LIN {X 0,Y 376.669,Z 402.869,A -85,B 0,C 180,E1 17335.147,E2 17335.147} C_VEL
LIN {X 0,Y 377.645,Z 382.714,A -85,B 0,C 180,E1 17334.66,E2 17334.66} C_VEL
LIN {X 0,Y 382.7,Z 216.459,A -85,B 0,C 180,E1 17331.601,E2 17331.601} C_VEL
LIN {X 0,Y 379.603,Z 196.687,A -85,B 0,C 180,E1 17330.72,E2 17330.72} C_VEL
LIN {X 0,Y 369.544,Z 178.657,A -85,B 0,C 180,E1 17328.838,E2 17328.838} C_VEL
LIN {X 0,Y 365.647,Z 171.977,A -85,B 0,C 180,E1 17328.055,E2 17328.055} C_VEL
LIN {X 0,Y 359.948,Z 157.351,A -85,B 0,C 180,E1 17324.899,E2 17324.899} C_VEL
LIN {X 0,Y 355.879,Z 147.74,A -85,B 0,C 180,E1 17322.598,E2 17322.598} C_VEL
LIN {X 0,Y 354.37,Z 147.289,A -85,B 0,C 180,E1 17322.197,E2 17322.197} C_VEL
LIN {X 0,Y 362.274,Z 168.365,A -85,B 0,C 180,E1 17319.144,E2 17319.144} C_VEL
LIN {X 0,Y 367.234,Z 183.559,A -85,B 0,C 180,E1 17317.084,E2 17317.084} C_VEL
LIN {X 0,Y 367.044,Z 189.046,A -85,B 0,C 180,E1 17316.607,E2 17316.607} C_VEL
LIN {X 0,Y 369.716,Z 213.655,A -85,B 0,C 180,E1 17315.636,E2 17315.636} C_VEL
LIN {X 0,Y 361.105,Z 400.958,A -85,B 0,C 180,E1 17310.874,E2 17310.874} C_VEL
LIN {X 0,Y 359.929,Z 421.052,A -85,B 0,C 180,E1 17310.048,E2 17310.048} C_VEL
LIN {X 0,Y 358.426,Z 440.427,A -85,B 0,C 180,E1 17308.947,E2 17308.947} C_VEL
LIN {X 0,Y 356.648,Z 459.281,A -85,B 0,C 180,E1 17307.554,E2 17307.554} C_VEL
LIN {X 0,Y 354.737,Z 477.04,A -85,B 0,C 180,E1 17305.905,E2 17305.905} C_VEL
LIN {X 0,Y 352.847,Z 493.012,A -85,B 0,C 180,E1 17304.083,E2 17304.083} C_VEL
LIN {X 0,Y 350.962,Z 507.993,A -85,B 0,C 180,E1 17302.002,E2 17302.002} C_VEL
LIN {X 0,Y 349.248,Z 521.455,A -85,B 0,C 180,E1 17299.745,E2 17299.745} C_VEL
LIN {X 0,Y 347.772,Z 533.32,A -85,B 0,C 180,E1 17297.345,E2 17297.345} C_VEL
LIN {X 0,Y 346.531,Z 544.028,A -85,B 0,C 180,E1 17294.709,E2 17294.709} C_VEL
LIN {X 0,Y 345.628,Z 552.855,A -85,B 0,C 180,E1 17292.022,E2 17292.022} C_VEL
LIN {X 0,Y 345.01,Z 560.233,A -85,B 0,C 180,E1 17289.172,E2 17289.172} C_VEL
LIN {X 0,Y 344.666,Z 565.763,A -85,B 0,C 180,E1 17286.329,E2 17286.329} C_VEL
LIN {X 0,Y 344.526,Z 569.587,A -85,B 0,C 180,E1 17283.494,E2 17283.494} C_VEL
LIN {X 0,Y 344.534,Z 571.796,A -85,B 0,C 180,E1 17280.665,E2 17280.665} C_VEL
LIN {X 0,Y 344.642,Z 572.453,A -85,B 0,C 180,E1 17277.839,E2 17277.839} C_VEL
LIN {X 0,Y 344.913,Z 571.551,A -85,B 0,C 180,E1 17275.011,E2 17275.011} C_VEL
LIN {X 0,Y 345.449,Z 568.896,A -85,B 0,C 180,E1 17272.014,E2 17272.014} C_VEL
LIN {X 0,Y 346.264,Z 564.713,A -85,B 0,C 180,E1 17269.182,E2 17269.182} C_VEL
LIN {X 0,Y 347.473,Z 558.782,A -85,B 0,C 180,E1 17266.352,E2 17266.352} C_VEL
LIN {X 0,Y 349.147,Z 550.97,A -85,B 0,C 180,E1 17263.531,E2 17263.531} C_VEL
LIN {X 0,Y 351.311,Z 540.92,A -85,B 0,C 180,E1 17260.723,E2 17260.723} C_VEL
LIN {X 0,Y 353.667,Z 529.913,A -85,B 0,C 180,E1 17258.263,E2 17258.263} C_VEL
LIN {X 0,Y 356.37,Z 517.049,A -85,B 0,C 180,E1 17255.907,E2 17255.907} C_VEL
LIN {X 0,Y 359.387,Z 501.97,A -85,B 0,C 180,E1 17253.657,E2 17253.657} C_VEL
LIN {X 0,Y 362.402,Z 485.474,A -85,B 0,C 180,E1 17251.671,E2 17251.671} C_VEL
LIN {X 0,Y 365.204,Z 468.627,A -85,B 0,C 180,E1 17250.023,E2 17250.023} C_VEL
LIN {X 0,Y 367.98,Z 450.12,A -85,B 0,C 180,E1 17248.554,E2 17248.554} C_VEL
LIN {X 0,Y 370.431,Z 430.981,A -85,B 0,C 180,E1 17247.368,E2 17247.368} C_VEL
LIN {X 0,Y 372.734,Z 409.425,A -85,B 0,C 180,E1 17246.363,E2 17246.363} C_VEL
LIN {X 0,Y 379.272,Z 352.203,A -85,B 0,C 180,E1 17244.383,E2 17244.383} C_VEL
LIN {X 0,Y 390.085,Z 279.328,A -85,B 0,C 180,E1 17241.833,E2 17241.833} C_VEL
LIN {X 0,Y 400.023,Z 222.705,A -85,B 0,C 180,E1 17239.855,E2 17239.855} C_VEL
LIN {X 0,Y 401.337,Z 211.185,A -85,B 0,C 180,E1 17238.798,E2 17238.798} C_VEL
LIN {X 0,Y 402.354,Z 207.214,A -85,B 0,C 180,E1 17238.338,E2 17238.338} C_VEL
LIN {X 0,Y 402.852,Z 202.964,A -85,B 0,C 180,E1 17236.862,E2 17236.862} C_VEL
LIN {X 0,Y 402.955,Z 202.336,A -85,B 0,C 180,E1 17236.432,E2 17236.432} C_VEL
LIN {X 0,Y 401.64,Z 206.111,A -85,B 0,C 180,E1 17235.499,E2 17235.499} C_VEL
LIN {X 0,Y 397.147,Z 221.02,A -85,B 0,C 180,E1 17234.85,E2 17234.85} C_VEL
LIN {X 0,Y 391.835,Z 244.614,A -85,B 0,C 180,E1 17234.018,E2 17234.018} C_VEL
LIN {X 0,Y 386.903,Z 267.436,A -85,B 0,C 180,E1 17233.236,E2 17233.236} C_VEL
LIN {X 0,Y 381.44,Z 294.492,A -85,B 0,C 180,E1 17232.25,E2 17232.25} C_VEL
LIN {X 0,Y 380.922,Z 302.139,A -85,B 0,C 180,E1 17232.058,E2 17232.058} C_VEL
LIN {X 0,Y 376.096,Z 417.535,A -85,B 0,C 180,E1 17229.641,E2 17229.641} C_VEL
LIN {X 0,Y 374.183,Z 439.175,A -85,B 0,C 180,E1 17228.934,E2 17228.934} C_VEL
LIN {X 0,Y 371.625,Z 460.279,A -85,B 0,C 180,E1 17227.947,E2 17227.947} C_VEL
LIN {X 0,Y 368.729,Z 479.932,A -85,B 0,C 180,E1 17226.722,E2 17226.722} C_VEL
LIN {X 0,Y 365.546,Z 498.613,A -85,B 0,C 180,E1 17225.25,E2 17225.25} C_VEL
LIN {X 0,Y 362.19,Z 516.529,A -85,B 0,C 180,E1 17223.513,E2 17223.513} C_VEL
LIN {X 0,Y 358.741,Z 533.822,A -85,B 0,C 180,E1 17221.476,E2 17221.476} C_VEL
LIN {X 0,Y 355.347,Z 550.311,A -85,B 0,C 180,E1 17219.13,E2 17219.13} C_VEL
LIN {X 0,Y 352.162,Z 565.804,A -85,B 0,C 180,E1 17216.473,E2 17216.473} C_VEL
LIN {X 0,Y 349.453,Z 579.625,A -85,B 0,C 180,E1 17213.615,E2 17213.615} C_VEL
LIN {X 0,Y 347.3,Z 591.834,A -85,B 0,C 180,E1 17210.564,E2 17210.564} C_VEL
LIN {X 0,Y 345.79,Z 601.923,A -85,B 0,C 180,E1 17207.502,E2 17207.502} C_VEL
LIN {X 0,Y 344.838,Z 610.17,A -85,B 0,C 180,E1 17204.436,E2 17204.436} C_VEL
LIN {X 0,Y 344.332,Z 616.936,A -85,B 0,C 180,E1 17201.22,E2 17201.22} C_VEL
LIN {X 0,Y 344.184,Z 621.714,A -85,B 0,C 180,E1 17198.185,E2 17198.185} C_VEL
LIN {X 0,Y 344.208,Z 625.148,A -85,B 0,C 180,E1 17195,E2 17195} C_VEL
LIN {X 0,Y 344.272,Z 626.894,A -85,B 0,C 180,E1 17191.998,E2 17191.998} C_VEL
LIN {X 0,Y 344.295,Z 627.095,A -85,B 0,C 180,E1 17189.003,E2 17189.003} C_VEL
LIN {X 0,Y 344.226,Z 625.768,A -85,B 0,C 180,E1 17185.837,E2 17185.837} C_VEL
LIN {X 0,Y 344.176,Z 623.016,A -85,B 0,C 180,E1 17182.825,E2 17182.825} C_VEL
LIN {X 0,Y 344.265,Z 618.402,A -85,B 0,C 180,E1 17179.627,E2 17179.627} C_VEL
LIN {X 0,Y 344.668,Z 611.955,A -85,B 0,C 180,E1 17176.363,E2 17176.363} C_VEL
LIN {X 0,Y 345.594,Z 603.383,A -85,B 0,C 180,E1 17173.011,E2 17173.011} C_VEL
LIN {X 0,Y 347.008,Z 593.607,A -85,B 0,C 180,E1 17169.938,E2 17169.938} C_VEL
LIN {X 0,Y 348.916,Z 582.559,A -85,B 0,C 180,E1 17167.064,E2 17167.064} C_VEL
LIN {X 0,Y 351.468,Z 569.316,A -85,B 0,C 180,E1 17164.2,E2 17164.2} C_VEL
LIN {X 0,Y 354.48,Z 554.472,A -85,B 0,C 180,E1 17161.532,E2 17161.532} C_VEL
LIN {X 0,Y 357.942,Z 537.753,A -85,B 0,C 180,E1 17159.043,E2 17159.043} C_VEL
LIN {X 0,Y 361.466,Z 520.196,A -85,B 0,C 180,E1 17156.887,E2 17156.887} C_VEL
LIN {X 0,Y 364.9,Z 502.06,A -85,B 0,C 180,E1 17155.064,E2 17155.064} C_VEL
LIN {X 0,Y 368.013,Z 483.999,A -85,B 0,C 180,E1 17153.585,E2 17153.585} C_VEL
LIN {X 0,Y 370.849,Z 465.441,A -85,B 0,C 180,E1 17152.363,E2 17152.363} C_VEL
LIN {X 0,Y 373.499,Z 444.639,A -85,B 0,C 180,E1 17151.307,E2 17151.307} C_VEL
LIN {X 0,Y 375.593,Z 423.414,A -85,B 0,C 180,E1 17150.54,E2 17150.54} C_VEL
LIN {X 0,Y 376.937,Z 399.024,A -85,B 0,C 180,E1 17149.951,E2 17149.951} C_VEL
LIN {X 0,Y 384.948,Z 202.452,A -85,B 0,C 180,E1 17145.917,E2 17145.917} C_VEL
LIN {X 0,Y 384.473,Z 199.885,A -85,B 0,C 180,E1 17145.79,E2 17145.79} C_VEL
LIN {X 0,Y 373.483,Z 180.271,A -85,B 0,C 180,E1 17143.765,E2 17143.765} C_VEL
LIN {X 0,Y 364.515,Z 165.595,A -85,B 0,C 180,E1 17141.984,E2 17141.984} C_VEL
LIN {X 0,Y 358.147,Z 151.33,A -85,B 0,C 180,E1 17138.913,E2 17138.913} C_VEL
LIN {X 0,Y 352.636,Z 139.889,A -85,B 0,C 180,E1 17136.14,E2 17136.14} C_VEL
LIN {X 0,Y 350.054,Z 135.087,A -85,B 0,C 180,E1 17134.838,E2 17134.838} C_VEL
LIN {X 0,Y 347.982,Z 130.852,A -85,B 0,C 180,E1 17133.679,E2 17133.679} C_VEL
LIN {X 0,Y 346.134,Z 127.573,A -85,B 0,C 180,E1 17132.695,E2 17132.695} C_VEL
LIN {X 0,Y 345.909,Z 126.377,A -85,B 0,C 180,E1 17132.38,E2 17132.38} C_VEL
LIN {X 0,Y 345.922,Z 126.373,A -85,B 0,C 180,E1 17128.17,E2 17128.17} C_VEL
LIN {X 0,Y 345.893,Z 126.372,A -85,B 0,C 180,E1 17123.871,E2 17123.871} C_VEL
LIN {X 0,Y 345.886,Z 126.376,A -85,B 0,C 180,E1 17119.768,E2 17119.768} C_VEL
LIN {X 0,Y 345.877,Z 126.4,A -85,B 0,C 180,E1 17115.595,E2 17115.595} C_VEL
LIN {X 0,Y 345.872,Z 126.388,A -85,B 0,C 180,E1 17111.337,E2 17111.337} C_VEL
LIN {X 0,Y 345.87,Z 126.366,A -85,B 0,C 180,E1 17107.14,E2 17107.14} C_VEL
LIN {X 0,Y 345.88,Z 126.39,A -85,B 0,C 180,E1 17102.982,E2 17102.982} C_VEL
LIN {X 0,Y 345.886,Z 126.391,A -85,B 0,C 180,E1 17098.84,E2 17098.84} C_VEL
LIN {X 0,Y 345.892,Z 126.363,A -85,B 0,C 180,E1 17094.692,E2 17094.692} C_VEL
LIN {X 0,Y 345.902,Z 126.39,A -85,B 0,C 180,E1 17090.516,E2 17090.516} C_VEL
LIN {X 0,Y 345.89,Z 126.392,A -85,B 0,C 180,E1 17086.227,E2 17086.227} C_VEL
LIN {X 0,Y 345.881,Z 126.368,A -85,B 0,C 180,E1 17082.156,E2 17082.156} C_VEL
LIN {X 0,Y 345.868,Z 126.38,A -85,B 0,C 180,E1 17077.925,E2 17077.925} C_VEL
LIN {X 0,Y 345.865,Z 126.4,A -85,B 0,C 180,E1 17073.657,E2 17073.657} C_VEL
LIN {X 0,Y 345.863,Z 126.401,A -85,B 0,C 180,E1 17069.416,E2 17069.416} C_VEL
LIN {X 0,Y 345.875,Z 126.395,A -85,B 0,C 180,E1 17065.182,E2 17065.182} C_VEL
LIN {X 0,Y 345.905,Z 126.617,A -85,B 0,C 180,E1 17063.193,E2 17063.193} C_VEL
LIN {X 0,Y 347.343,Z 130.105,A -85,B 0,C 180,E1 17062.183,E2 17062.183} C_VEL
LIN {X 0,Y 348.365,Z 132.049,A -85,B 0,C 180,E1 17061.585,E2 17061.585} C_VEL
LIN {X 0,Y 350.531,Z 136.549,A -85,B 0,C 180,E1 17060.287,E2 17060.287} C_VEL
LIN {X 0,Y 354.726,Z 145.516,A -85,B 0,C 180,E1 17057.867,E2 17057.867} C_VEL
LIN {X 0,Y 360.366,Z 158.402,A -85,B 0,C 180,E1 17054.741,E2 17054.741} C_VEL
LIN {X 0,Y 365.903,Z 172.565,A -85,B 0,C 180,E1 17051.755,E2 17051.755} C_VEL
LIN {X 0,Y 376.444,Z 190.872,A -85,B 0,C 180,E1 17049.742,E2 17049.742} C_VEL
LIN {X 0,Y 379.861,Z 197.758,A -85,B 0,C 180,E1 17049.104,E2 17049.104} C_VEL
LIN {X 0,Y 382.711,Z 218.275,A -85,B 0,C 180,E1 17048.246,E2 17048.246} C_VEL
LIN {X 0,Y 377.126,Z 394.489,A -85,B 0,C 180,E1 17044.986,E2 17044.986} C_VEL
LIN {X 0,Y 375.738,Z 413.928,A -85,B 0,C 180,E1 17044.359,E2 17044.359} C_VEL
LIN {X 0,Y 373.878,Z 431.784,A -85,B 0,C 180,E1 17043.52,E2 17043.52} C_VEL
LIN {X 0,Y 371.403,Z 449.716,A -85,B 0,C 180,E1 17042.392,E2 17042.392} C_VEL
LIN {X 0,Y 368.525,Z 466.63,A -85,B 0,C 180,E1 17041.029,E2 17041.029} C_VEL
LIN {X 0,Y 365.237,Z 483.324,A -85,B 0,C 180,E1 17039.341,E2 17039.341} C_VEL
LIN {X 0,Y 361.781,Z 498.814,A -85,B 0,C 180,E1 17037.396,E2 17037.396} C_VEL
LIN {X 0,Y 358.417,Z 512.658,A -85,B 0,C 180,E1 17035.264,E2 17035.264} C_VEL
LIN {X 0,Y 355.163,Z 525.427,A -85,B 0,C 180,E1 17032.86,E2 17032.86} C_VEL
LIN {X 0,Y 352.22,Z 536.673,A -85,B 0,C 180,E1 17030.261,E2 17030.261} C_VEL
LIN {X 0,Y 349.57,Z 546.939,A -85,B 0,C 180,E1 17027.304,E2 17027.304} C_VEL
LIN {X 0,Y 347.575,Z 555.103,A -85,B 0,C 180,E1 17024.322,E2 17024.322} C_VEL
LIN {X 0,Y 346.111,Z 561.733,A -85,B 0,C 180,E1 17021.159,E2 17021.159} C_VEL
LIN {X 0,Y 345.205,Z 566.551,A -85,B 0,C 180,E1 17017.99,E2 17017.99} C_VEL
LIN {X 0,Y 344.718,Z 569.704,A -85,B 0,C 180,E1 17014.824,E2 17014.824} C_VEL
LIN {X 0,Y 344.514,Z 571.318,A -85,B 0,C 180,E1 17011.496,E2 17011.496} C_VEL
LIN {X 0,Y 344.523,Z 571.26,A -85,B 0,C 180,E1 17008.17,E2 17008.17} C_VEL
LIN {X 0,Y 344.742,Z 569.524,A -85,B 0,C 180,E1 17004.841,E2 17004.841} C_VEL
LIN {X 0,Y 345.047,Z 567.492,A -85,B 0,C 180,E1 17002.726,E2 17002.726} C_VEL
LIN {X 0,Y 344.31,Z 566.093,A -85,B 0,C 180,E1 17001.465,E2 17001.465} C_VEL
LIN {X 0,Y 339.153,Z 561.593,A -85,B 0,C 180,E1 16998.087,E2 16998.087} C_VEL
LIN {X 0,Y 338.885,Z 559.609,A -85,B 0,C 180,E1 16997.007,E2 16997.007} C_VEL
LIN {X 0,Y 340.728,Z 552.186,A -85,B 0,C 180,E1 16993.812,E2 16993.812} C_VEL
LIN {X 0,Y 343.148,Z 543.092,A -85,B 0,C 180,E1 16990.775,E2 16990.775} C_VEL
LIN {X 0,Y 346.088,Z 532.413,A -85,B 0,C 180,E1 16987.939,E2 16987.939} C_VEL
LIN {X 0,Y 349.449,Z 520.13,A -85,B 0,C 180,E1 16985.307,E2 16985.307} C_VEL
LIN {X 0,Y 352.96,Z 506.734,A -85,B 0,C 180,E1 16982.974,E2 16982.974} C_VEL
LIN {X 0,Y 356.567,Z 492.027,A -85,B 0,C 180,E1 16980.887,E2 16980.887} C_VEL
LIN {X 0,Y 360.18,Z 475.636,A -85,B 0,C 180,E1 16979.005,E2 16979.005} C_VEL
LIN {X 0,Y 363.415,Z 458.807,A -85,B 0,C 180,E1 16977.46,E2 16977.46} C_VEL
LIN {X 0,Y 366.3,Z 440.809,A -85,B 0,C 180,E1 16976.161,E2 16976.161} C_VEL
LIN {X 0,Y 368.645,Z 422.047,A -85,B 0,C 180,E1 16975.137,E2 16975.137} C_VEL
LIN {X 0,Y 370.332,Z 403.037,A -85,B 0,C 180,E1 16974.396,E2 16974.396} C_VEL
LIN {X 0,Y 371.349,Z 382.958,A -85,B 0,C 180,E1 16973.905,E2 16973.905} C_VEL
LIN {X 0,Y 376.667,Z 217.846,A -85,B 0,C 180,E1 16970.825,E2 16970.825} C_VEL
LIN {X 0,Y 374.047,Z 200.618,A -85,B 0,C 180,E1 16970.042,E2 16970.042} C_VEL
LIN {X 0,Y 363.82,Z 182.148,A -85,B 0,C 180,E1 16968.051,E2 16968.051} C_VEL
LIN {X 0,Y 357.676,Z 171.867,A -85,B 0,C 180,E1 16966.773,E2 16966.773} C_VEL
LIN {X 0,Y 351.569,Z 156.622,A -85,B 0,C 180,E1 16963.268,E2 16963.268} C_VEL
LIN {X 0,Y 350.226,Z 154.037,A -85,B 0,C 180,E1 16962.58,E2 16962.58} C_VEL
LIN {X 0,Y 348.669,Z 153.653,A -85,B 0,C 180,E1 16962.158,E2 16962.158} C_VEL
LIN {X 0,Y 356.203,Z 174.193,A -85,B 0,C 180,E1 16959.167,E2 16959.167} C_VEL
LIN {X 0,Y 360.109,Z 185.882,A -85,B 0,C 180,E1 16957.56,E2 16957.56} C_VEL
LIN {X 0,Y 360.055,Z 189.639,A -85,B 0,C 180,E1 16957.242,E2 16957.242} C_VEL
LIN {X 0,Y 362.693,Z 214.583,A -85,B 0,C 180,E1 16956.227,E2 16956.227} C_VEL
LIN {X 0,Y 353.679,Z 401.543,A -85,B 0,C 180,E1 16951.344,E2 16951.344} C_VEL
LIN {X 0,Y 352.479,Z 421.326,A -85,B 0,C 180,E1 16950.515,E2 16950.515} C_VEL
LIN {X 0,Y 350.98,Z 440.119,A -85,B 0,C 180,E1 16949.434,E2 16949.434} C_VEL
LIN {X 0,Y 349.131,Z 459.141,A -85,B 0,C 180,E1 16948.013,E2 16948.013} C_VEL
LIN {X 0,Y 347.255,Z 476.075,A -85,B 0,C 180,E1 16946.43,E2 16946.43} C_VEL
LIN {X 0,Y 345.316,Z 492.049,A -85,B 0,C 180,E1 16944.605,E2 16944.605} C_VEL
LIN {X 0,Y 343.374,Z 507.168,A -85,B 0,C 180,E1 16942.514,E2 16942.514} C_VEL
LIN {X 0,Y 341.566,Z 520.911,A -85,B 0,C 180,E1 16940.208,E2 16940.208} C_VEL
LIN {X 0,Y 340.033,Z 532.774,A -85,B 0,C 180,E1 16937.807,E2 16937.807} C_VEL
LIN {X 0,Y 338.725,Z 543.603,A -85,B 0,C 180,E1 16935.146,E2 16935.146} C_VEL
LIN {X 0,Y 337.728,Z 552.932,A -85,B 0,C 180,E1 16932.308,E2 16932.308} C_VEL
LIN {X 0,Y 337.065,Z 560.461,A -85,B 0,C 180,E1 16929.39,E2 16929.39} C_VEL
LIN {X 0,Y 336.697,Z 566.123,A -85,B 0,C 180,E1 16926.48,E2 16926.48} C_VEL
LIN {X 0,Y 336.547,Z 570.075,A -85,B 0,C 180,E1 16923.577,E2 16923.577} C_VEL
LIN {X 0,Y 336.558,Z 572.419,A -85,B 0,C 180,E1 16920.681,E2 16920.681} C_VEL
LIN {X 0,Y 336.679,Z 573.197,A -85,B 0,C 180,E1 16917.788,E2 16917.788} C_VEL
LIN {X 0,Y 336.979,Z 572.412,A -85,B 0,C 180,E1 16914.893,E2 16914.893} C_VEL
LIN {X 0,Y 337.566,Z 569.88,A -85,B 0,C 180,E1 16911.827,E2 16911.827} C_VEL
LIN {X 0,Y 338.522,Z 565.528,A -85,B 0,C 180,E1 16908.759,E2 16908.759} C_VEL
LIN {X 0,Y 339.865,Z 559.637,A -85,B 0,C 180,E1 16905.867,E2 16905.867} C_VEL
LIN {X 0,Y 341.702,Z 551.853,A -85,B 0,C 180,E1 16902.986,E2 16902.986} C_VEL
LIN {X 0,Y 343.909,Z 542.508,A -85,B 0,C 180,E1 16900.291,E2 16900.291} C_VEL
LIN {X 0,Y 346.448,Z 531.764,A -85,B 0,C 180,E1 16897.786,E2 16897.786} C_VEL
LIN {X 0,Y 349.439,Z 518.656,A -85,B 0,C 180,E1 16895.307,E2 16895.307} C_VEL
LIN {X 0,Y 352.669,Z 503.818,A -85,B 0,C 180,E1 16893.024,E2 16893.024} C_VEL
LIN {X 0,Y 355.777,Z 488.46,A -85,B 0,C 180,E1 16891.094,E2 16891.094} C_VEL
LIN {X 0,Y 358.924,Z 471.463,A -85,B 0,C 180,E1 16889.351,E2 16889.351} C_VEL
LIN {X 0,Y 362.057,Z 452.668,A -85,B 0,C 180,E1 16887.793,E2 16887.793} C_VEL
LIN {X 0,Y 364.883,Z 433.34,A -85,B 0,C 180,E1 16886.532,E2 16886.532} C_VEL
LIN {X 0,Y 367.478,Z 411.855,A -85,B 0,C 180,E1 16885.479,E2 16885.479} C_VEL
LIN {X 0,Y 374.158,Z 359.163,A -85,B 0,C 180,E1 16883.577,E2 16883.577} C_VEL
LIN {X 0,Y 385.505,Z 288.757,A -85,B 0,C 180,E1 16881.051,E2 16881.051} C_VEL
LIN {X 0,Y 397.659,Z 225.322,A -85,B 0,C 180,E1 16878.807,E2 16878.807} C_VEL
LIN {X 0,Y 399.563,Z 213.082,A -85,B 0,C 180,E1 16877.631,E2 16877.631} C_VEL
LIN {X 0,Y 400.105,Z 210.398,A -85,B 0,C 180,E1 16876.607,E2 16876.607} C_VEL
LIN {X 0,Y 399.764,Z 211.263,A -85,B 0,C 180,E1 16876.445,E2 16876.445} C_VEL
LIN {X 0,Y 396.708,Z 221.504,A -85,B 0,C 180,E1 16876.033,E2 16876.033} C_VEL
LIN {X 0,Y 389.126,Z 252.716,A -85,B 0,C 180,E1 16874.961,E2 16874.961} C_VEL
LIN {X 0,Y 383.159,Z 278.56,A -85,B 0,C 180,E1 16874.05,E2 16874.05} C_VEL
LIN {X 0,Y 377.866,Z 302.725,A -85,B 0,C 180,E1 16873.172,E2 16873.172} C_VEL
LIN {X 0,Y 373.832,Z 323.539,A -85,B 0,C 180,E1 16872.388,E2 16872.388} C_VEL
LIN {X 0,Y 369.736,Z 417.309,A -85,B 0,C 180,E1 16870.392,E2 16870.392} C_VEL
LIN {X 0,Y 367.763,Z 438.86,A -85,B 0,C 180,E1 16869.68,E2 16869.68} C_VEL
LIN {X 0,Y 365.152,Z 459.562,A -85,B 0,C 180,E1 16868.704,E2 16868.704} C_VEL
LIN {X 0,Y 362.026,Z 479.974,A -85,B 0,C 180,E1 16867.418,E2 16867.418} C_VEL
LIN {X 0,Y 358.545,Z 499.478,A -85,B 0,C 180,E1 16865.848,E2 16865.848} C_VEL
LIN {X 0,Y 354.905,Z 517.907,A -85,B 0,C 180,E1 16864.003,E2 16864.003} C_VEL
LIN {X 0,Y 351.368,Z 534.672,A -85,B 0,C 180,E1 16861.958,E2 16861.958} C_VEL
LIN {X 0,Y 347.911,Z 550.579,A -85,B 0,C 180,E1 16859.625,E2 16859.625} C_VEL
LIN {X 0,Y 344.755,Z 565.071,A -85,B 0,C 180,E1 16857.082,E2 16857.082} C_VEL
LIN {X 0,Y 341.855,Z 579.016,A -85,B 0,C 180,E1 16854.142,E2 16854.142} C_VEL
LIN {X 0,Y 339.553,Z 591.234,A -85,B 0,C 180,E1 16851.022,E2 16851.022} C_VEL
LIN {X 0,Y 337.943,Z 601.228,A -85,B 0,C 180,E1 16847.922,E2 16847.922} C_VEL
LIN {X 0,Y 336.878,Z 609.823,A -85,B 0,C 180,E1 16844.632,E2 16844.632} C_VEL
LIN {X 0,Y 336.343,Z 616.593,A -85,B 0,C 180,E1 16841.316,E2 16841.316} C_VEL
LIN {X 0,Y 336.193,Z 621.506,A -85,B 0,C 180,E1 16838.036,E2 16838.036} C_VEL
LIN {X 0,Y 336.232,Z 624.749,A -85,B 0,C 180,E1 16834.777,E2 16834.777} C_VEL
LIN {X 0,Y 336.303,Z 626.347,A -85,B 0,C 180,E1 16831.705,E2 16831.705} C_VEL
LIN {X 0,Y 336.317,Z 626.424,A -85,B 0,C 180,E1 16828.809,E2 16828.809} C_VEL
LIN {X 0,Y 336.24,Z 624.994,A -85,B 0,C 180,E1 16825.567,E2 16825.567} C_VEL
LIN {X 0,Y 336.187,Z 622.17,A -85,B 0,C 180,E1 16822.482,E2 16822.482} C_VEL
LIN {X 0,Y 336.301,Z 617.458,A -85,B 0,C 180,E1 16819.206,E2 16819.206} C_VEL
LIN {X 0,Y 336.755,Z 611,A -85,B 0,C 180,E1 16815.91,E2 16815.91} C_VEL
LIN {X 0,Y 337.734,Z 602.686,A -85,B 0,C 180,E1 16812.603,E2 16812.603} C_VEL
LIN {X 0,Y 339.356,Z 592.318,A -85,B 0,C 180,E1 16809.296,E2 16809.296} C_VEL
LIN {X 0,Y 341.442,Z 581.082,A -85,B 0,C 180,E1 16806.349,E2 16806.349} C_VEL
LIN {X 0,Y 344.14,Z 567.986,A -85,B 0,C 180,E1 16803.49,E2 16803.49} C_VEL
LIN {X 0,Y 347.337,Z 553.164,A -85,B 0,C 180,E1 16800.797,E2 16800.797} C_VEL
LIN {X 0,Y 350.834,Z 537.114,A -85,B 0,C 180,E1 16798.374,E2 16798.374} C_VEL
LIN {X 0,Y 354.597,Z 519.321,A -85,B 0,C 180,E1 16796.16,E2 16796.16} C_VEL
LIN {X 0,Y 358.364,Z 500.272,A -85,B 0,C 180,E1 16794.233,E2 16794.233} C_VEL
LIN {X 0,Y 361.828,Z 480.911,A -85,B 0,C 180,E1 16792.661,E2 16792.661} C_VEL
LIN {X 0,Y 364.803,Z 461.647,A -85,B 0,C 180,E1 16791.427,E2 16791.427} C_VEL
LIN {X 0,Y 367.379,Z 441.543,A -85,B 0,C 180,E1 16790.444,E2 16790.444} C_VEL
LIN {X 0,Y 369.386,Z 421.025,A -85,B 0,C 180,E1 16789.727,E2 16789.727} C_VEL
LIN {X 0,Y 370.89,Z 392.105,A -85,B 0,C 180,E1 16789.055,E2 16789.055} C_VEL
LIN {X 0,Y 378.87,Z 203.932,A -85,B 0,C 180,E1 16785.146,E2 16785.146} C_VEL
LIN {X 0,Y 368.573,Z 185.369,A -85,B 0,C 180,E1 16783.18,E2 16783.18} C_VEL
LIN {X 0,Y 358.66,Z 169.273,A -85,B 0,C 180,E1 16781.167,E2 16781.167} C_VEL
LIN {X 0,Y 356.331,Z 165.47,A -85,B 0,C 180,E1 16780.616,E2 16780.616} C_VEL
LIN {X 0,Y 350.756,Z 153.122,A -85,B 0,C 180,E1 16777.797,E2 16777.797} C_VEL
LIN {X 0,Y 345.132,Z 141.448,A -85,B 0,C 180,E1 16774.8,E2 16774.8} C_VEL
LIN {X 0,Y 342.33,Z 136.309,A -85,B 0,C 180,E1 16773.305,E2 16773.305} C_VEL
LIN {X 0,Y 340.529,Z 132.462,A -85,B 0,C 180,E1 16772.203,E2 16772.203} C_VEL
LIN {X 0,Y 338.247,Z 128.784,A -85,B 0,C 180,E1 16770.953,E2 16770.953} C_VEL
LIN {X 0,Y 337.961,Z 127.386,A -85,B 0,C 180,E1 16770.582,E2 16770.582} C_VEL
LIN {X 0,Y 337.974,Z 127.388,A -85,B 0,C 180,E1 16766.315,E2 16766.315} C_VEL
LIN {X 0,Y 337.97,Z 127.379,A -85,B 0,C 180,E1 16762.068,E2 16762.068} C_VEL
LIN {X 0,Y 337.944,Z 127.364,A -85,B 0,C 180,E1 16757.742,E2 16757.742} C_VEL
LIN {X 0,Y 337.934,Z 127.356,A -85,B 0,C 180,E1 16753.517,E2 16753.517} C_VEL
LIN {X 0,Y 337.935,Z 127.38,A -85,B 0,C 180,E1 16749.193,E2 16749.193} C_VEL
LIN {X 0,Y 337.944,Z 127.383,A -85,B 0,C 180,E1 16744.922,E2 16744.922} C_VEL
LIN {X 0,Y 337.962,Z 127.35,A -85,B 0,C 180,E1 16740.593,E2 16740.593} C_VEL
LIN {X 0,Y 337.96,Z 127.372,A -85,B 0,C 180,E1 16736.438,E2 16736.438} C_VEL
LIN {X 0,Y 337.952,Z 127.383,A -85,B 0,C 180,E1 16732.178,E2 16732.178} C_VEL
LIN {X 0,Y 337.932,Z 127.357,A -85,B 0,C 180,E1 16727.873,E2 16727.873} C_VEL
LIN {X 0,Y 337.926,Z 127.368,A -85,B 0,C 180,E1 16723.675,E2 16723.675} C_VEL
LIN {X 0,Y 337.93,Z 127.391,A -85,B 0,C 180,E1 16719.384,E2 16719.384} C_VEL
LIN {X 0,Y 337.934,Z 127.373,A -85,B 0,C 180,E1 16715.156,E2 16715.156} C_VEL
LIN {X 0,Y 337.945,Z 127.36,A -85,B 0,C 180,E1 16710.973,E2 16710.973} C_VEL
LIN {X 0,Y 337.951,Z 127.362,A -85,B 0,C 180,E1 16706.815,E2 16706.815} C_VEL
LIN {X 0,Y 337.979,Z 127.626,A -85,B 0,C 180,E1 16704.976,E2 16704.976} C_VEL
LIN {X 0,Y 339.396,Z 131.102,A -85,B 0,C 180,E1 16703.899,E2 16703.899} C_VEL
LIN {X 0,Y 340.451,Z 132.811,A -85,B 0,C 180,E1 16703.297,E2 16703.297} C_VEL
LIN {X 0,Y 344.764,Z 141.822,A -85,B 0,C 180,E1 16700.57,E2 16700.57} C_VEL
LIN {X 0,Y 349.842,Z 152.762,A -85,B 0,C 180,E1 16697.585,E2 16697.585} C_VEL
LIN {X 0,Y 355.683,Z 166.992,A -85,B 0,C 180,E1 16694.197,E2 16694.197} C_VEL
LIN {X 0,Y 357.902,Z 172.461,A -85,B 0,C 180,E1 16693.038,E2 16693.038} C_VEL
LIN {X 0,Y 368.613,Z 190.696,A -85,B 0,C 180,E1 16690.877,E2 16690.877} C_VEL
LIN {X 0,Y 374.224,Z 201.393,A -85,B 0,C 180,E1 16689.797,E2 16689.797} C_VEL
LIN {X 0,Y 376.663,Z 219.69,A -85,B 0,C 180,E1 16689.02,E2 16689.02} C_VEL
LIN {X 0,Y 370.794,Z 394.883,A -85,B 0,C 180,E1 16685.733,E2 16685.733} C_VEL
LIN {X 0,Y 369.349,Z 414.285,A -85,B 0,C 180,E1 16685.098,E2 16685.098} C_VEL
LIN {X 0,Y 367.3,Z 432.961,A -85,B 0,C 180,E1 16684.202,E2 16684.202} C_VEL
LIN {X 0,Y 364.727,Z 450.731,A -85,B 0,C 180,E1 16683.06,E2 16683.06} C_VEL
LIN {X 0,Y 361.572,Z 468.366,A -85,B 0,C 180,E1 16681.601,E2 16681.601} C_VEL
LIN {X 0,Y 358.159,Z 484.804,A -85,B 0,C 180,E1 16679.887,E2 16679.887} C_VEL
LIN {X 0,Y 354.57,Z 500.118,A -85,B 0,C 180,E1 16677.91,E2 16677.91} C_VEL
LIN {X 0,Y 351.2,Z 513.393,A -85,B 0,C 180,E1 16675.821,E2 16675.821} C_VEL
LIN {X 0,Y 347.793,Z 526.134,A -85,B 0,C 180,E1 16673.373,E2 16673.373} C_VEL
LIN {X 0,Y 344.705,Z 537.363,A -85,B 0,C 180,E1 16670.723,E2 16670.723} C_VEL
LIN {X 0,Y 342.053,Z 547.116,A -85,B 0,C 180,E1 16667.873,E2 16667.873} C_VEL
LIN {X 0,Y 339.906,Z 555.38,A -85,B 0,C 180,E1 16664.827,E2 16664.827} C_VEL
LIN {X 0,Y 338.317,Z 562.106,A -85,B 0,C 180,E1 16661.592,E2 16661.592} C_VEL
LIN {X 0,Y 337.323,Z 567.008,A -85,B 0,C 180,E1 16658.35,E2 16658.35} C_VEL
LIN {X 0,Y 336.76,Z 570.351,A -85,B 0,C 180,E1 16654.938,E2 16654.938} C_VEL
LIN {X 0,Y 336.541,Z 571.964,A -85,B 0,C 180,E1 16651.531,E2 16651.531} C_VEL
LIN {X 0,Y 336.551,Z 571.905,A -85,B 0,C 180,E1 16648.126,E2 16648.126} C_VEL
LIN {X 0,Y 336.787,Z 570.171,A -85,B 0,C 180,E1 16644.718,E2 16644.718} C_VEL
LIN {X 0,Y 337.344,Z 566.922,A -85,B 0,C 180,E1 16641.477,E2 16641.477} C_VEL
LIN {X 0,Y 338.42,Z 561.658,A -85,B 0,C 180,E1 16638.063,E2 16638.063} C_VEL
LIN {X 0,Y 338.885,Z 559.609,A -85,B 0,C 180,E1 16637.007,E2 16637.007} C_VEL
LIN {X 0,Y 338.544,Z 557.217,A -85,B 0,C 180,E1 16635.758,E2 16635.758} C_VEL
LIN {X 0,Y 334.79,Z 550.945,A -85,B 0,C 180,E1 16632.765,E2 16632.765} C_VEL
LIN {X 0,Y 334.502,Z 547.665,A -85,B 0,C 180,E1 16631.558,E2 16631.558} C_VEL
LIN {X 0,Y 334.618,Z 547.147,A -85,B 0,C 180,E1 16631.391,E2 16631.391} C_VEL
LIN {X 0,Y 337.5,Z 537.117,A -85,B 0,C 180,E1 16628.446,E2 16628.446} C_VEL
LIN {X 0,Y 340.799,Z 525.71,A -85,B 0,C 180,E1 16625.748,E2 16625.748} C_VEL
LIN {X 0,Y 344.423,Z 512.758,A -85,B 0,C 180,E1 16623.258,E2 16623.258} C_VEL
LIN {X 0,Y 348.132,Z 498.713,A -85,B 0,C 180,E1 16621.056,E2 16621.056} C_VEL
LIN {X 0,Y 351.771,Z 483.716,A -85,B 0,C 180,E1 16619.137,E2 16619.137} C_VEL
LIN {X 0,Y 355.2,Z 467.72,A -85,B 0,C 180,E1 16617.475,E2 16617.475} C_VEL
LIN {X 0,Y 358.319,Z 450.85,A -85,B 0,C 180,E1 16616.076,E2 16616.076} C_VEL
LIN {X 0,Y 361.089,Z 432.312,A -85,B 0,C 180,E1 16614.881,E2 16614.881} C_VEL
LIN {X 0,Y 363.233,Z 413.203,A -85,B 0,C 180,E1 16613.975,E2 16613.975} C_VEL
LIN {X 0,Y 364.676,Z 393.727,A -85,B 0,C 180,E1 16613.351,E2 16613.351} C_VEL
LIN {X 0,Y 370.694,Z 219.152,A -85,B 0,C 180,E1 16610.02,E2 16610.02} C_VEL
LIN {X 0,Y 368.466,Z 204.357,A -85,B 0,C 180,E1 16609.328,E2 16609.328} C_VEL
LIN {X 0,Y 358.773,Z 186.808,A -85,B 0,C 180,E1 16607.37,E2 16607.37} C_VEL
LIN {X 0,Y 349.655,Z 171.823,A -85,B 0,C 180,E1 16605.401,E2 16605.401} C_VEL
LIN {X 0,Y 345.002,Z 160.411,A -85,B 0,C 180,E1 16602.644,E2 16602.644} C_VEL
LIN {X 0,Y 342.949,Z 160.049,A -85,B 0,C 180,E1 16602.129,E2 16602.129} C_VEL
LIN {X 0,Y 350.82,Z 182.032,A -85,B 0,C 180,E1 16598.915,E2 16598.915} C_VEL
LIN {X 0,Y 352.984,Z 189.385,A -85,B 0,C 180,E1 16597.929,E2 16597.929} C_VEL
LIN {X 0,Y 355.682,Z 215.64,A -85,B 0,C 180,E1 16596.832,E2 16596.832} C_VEL
LIN {X 0,Y 346.28,Z 402.045,A -85,B 0,C 180,E1 16591.837,E2 16591.837} C_VEL
LIN {X 0,Y 345.051,Z 421.535,A -85,B 0,C 180,E1 16591.002,E2 16591.002} C_VEL
LIN {X 0,Y 343.436,Z 440.963,A -85,B 0,C 180,E1 16589.858,E2 16589.858} C_VEL
LIN {X 0,Y 341.525,Z 459.91,A -85,B 0,C 180,E1 16588.408,E2 16588.408} C_VEL
LIN {X 0,Y 339.481,Z 477.701,A -85,B 0,C 180,E1 16586.698,E2 16586.698} C_VEL
LIN {X 0,Y 337.443,Z 493.872,A -85,B 0,C 180,E1 16584.789,E2 16584.789} C_VEL
LIN {X 0,Y 335.419,Z 508.971,A -85,B 0,C 180,E1 16582.616,E2 16582.616} C_VEL
LIN {X 0,Y 333.569,Z 522.585,A -85,B 0,C 180,E1 16580.246,E2 16580.246} C_VEL
LIN {X 0,Y 331.972,Z 534.637,A -85,B 0,C 180,E1 16577.71,E2 16577.71} C_VEL
LIN {X 0,Y 330.628,Z 545.593,A -85,B 0,C 180,E1 16574.895,E2 16574.895} C_VEL
LIN {X 0,Y 329.676,Z 554.43,A -85,B 0,C 180,E1 16572.08,E2 16572.08} C_VEL
LIN {X 0,Y 329.062,Z 561.418,A -85,B 0,C 180,E1 16569.268,E2 16569.268} C_VEL
LIN {X 0,Y 328.7,Z 567.047,A -85,B 0,C 180,E1 16566.287,E2 16566.287} C_VEL
LIN {X 0,Y 328.564,Z 570.955,A -85,B 0,C 180,E1 16563.315,E2 16563.315} C_VEL
LIN {X 0,Y 328.592,Z 573.238,A -85,B 0,C 180,E1 16560.349,E2 16560.349} C_VEL
LIN {X 0,Y 328.747,Z 573.957,A -85,B 0,C 180,E1 16557.386,E2 16557.386} C_VEL
LIN {X 0,Y 329.102,Z 573.112,A -85,B 0,C 180,E1 16554.421,E2 16554.421} C_VEL
LIN {X 0,Y 329.786,Z 570.519,A -85,B 0,C 180,E1 16551.281,E2 16551.281} C_VEL
LIN {X 0,Y 330.806,Z 566.392,A -85,B 0,C 180,E1 16548.317,E2 16548.317} C_VEL
LIN {X 0,Y 332.399,Z 560.161,A -85,B 0,C 180,E1 16545.186,E2 16545.186} C_VEL
LIN {X 0,Y 334.433,Z 552.267,A -85,B 0,C 180,E1 16542.245,E2 16542.245} C_VEL
LIN {X 0,Y 336.881,Z 542.901,A -85,B 0,C 180,E1 16539.499,E2 16539.499} C_VEL
LIN {X 0,Y 339.865,Z 531.302,A -85,B 0,C 180,E1 16536.783,E2 16536.783} C_VEL
LIN {X 0,Y 343.17,Z 518.029,A -85,B 0,C 180,E1 16534.271,E2 16534.271} C_VEL
LIN {X 0,Y 346.449,Z 504.168,A -85,B 0,C 180,E1 16532.126,E2 16532.126} C_VEL
LIN {X 0,Y 349.964,Z 488.184,A -85,B 0,C 180,E1 16530.096,E2 16530.096} C_VEL
LIN {X 0,Y 353.565,Z 470.437,A -85,B 0,C 180,E1 16528.265,E2 16528.265} C_VEL
LIN {X 0,Y 356.827,Z 452.695,A -85,B 0,C 180,E1 16526.784,E2 16526.784} C_VEL
LIN {X 0,Y 359.803,Z 434.285,A -85,B 0,C 180,E1 16525.563,E2 16525.563} C_VEL
LIN {X 0,Y 362.703,Z 413.184,A -85,B 0,C 180,E1 16524.494,E2 16524.494} C_VEL
LIN {X 0,Y 369.845,Z 362.804,A -85,B 0,C 180,E1 16522.609,E2 16522.609} C_VEL
LIN {X 0,Y 382.563,Z 291.283,A -85,B 0,C 180,E1 16519.989,E2 16519.989} C_VEL
LIN {X 0,Y 395.791,Z 228.046,A -85,B 0,C 180,E1 16517.737,E2 16517.737} C_VEL
LIN {X 0,Y 396.766,Z 222.549,A -85,B 0,C 180,E1 16517.193,E2 16517.193} C_VEL
LIN {X 0,Y 388.461,Z 254.303,A -85,B 0,C 180,E1 16516.113,E2 16516.113} C_VEL
LIN {X 0,Y 381.886,Z 280.576,A -85,B 0,C 180,E1 16515.198,E2 16515.198} C_VEL
LIN {X 0,Y 376.194,Z 304.392,A -85,B 0,C 180,E1 16514.335,E2 16514.335} C_VEL
LIN {X 0,Y 370.732,Z 328.655,A -85,B 0,C 180,E1 16513.439,E2 16513.439} C_VEL
LIN {X 0,Y 366.675,Z 347.809,A -85,B 0,C 180,E1 16512.685,E2 16512.685} C_VEL
LIN {X 0,Y 363.403,Z 417.556,A -85,B 0,C 180,E1 16511.156,E2 16511.156} C_VEL
LIN {X 0,Y 361.383,Z 438.754,A -85,B 0,C 180,E1 16510.443,E2 16510.443} C_VEL
LIN {X 0,Y 358.627,Z 459.706,A -85,B 0,C 180,E1 16509.441,E2 16509.441} C_VEL
LIN {X 0,Y 355.463,Z 479.493,A -85,B 0,C 180,E1 16508.176,E2 16508.176} C_VEL
LIN {X 0,Y 351.929,Z 498.508,A -85,B 0,C 180,E1 16506.63,E2 16506.63} C_VEL
LIN {X 0,Y 348.264,Z 516.264,A -85,B 0,C 180,E1 16504.844,E2 16504.844} C_VEL
LIN {X 0,Y 344.531,Z 533.215,A -85,B 0,C 180,E1 16502.769,E2 16502.769} C_VEL
LIN {X 0,Y 340.894,Z 549.118,A -85,B 0,C 180,E1 16500.423,E2 16500.423} C_VEL
LIN {X 0,Y 337.404,Z 564.293,A -85,B 0,C 180,E1 16497.728,E2 16497.728} C_VEL
LIN {X 0,Y 334.504,Z 577.424,A -85,B 0,C 180,E1 16494.928,E2 16494.928} C_VEL
LIN {X 0,Y 332.108,Z 589.193,A -85,B 0,C 180,E1 16491.922,E2 16491.922} C_VEL
LIN {X 0,Y 330.275,Z 599.55,A -85,B 0,C 180,E1 16488.718,E2 16488.718} C_VEL
LIN {X 0,Y 329.049,Z 608.371,A -85,B 0,C 180,E1 16485.33,E2 16485.33} C_VEL
LIN {X 0,Y 328.411,Z 615.266,A -85,B 0,C 180,E1 16481.949,E2 16481.949} C_VEL
LIN {X 0,Y 328.206,Z 620.396,A -85,B 0,C 180,E1 16478.586,E2 16478.586} C_VEL
LIN {X 0,Y 328.239,Z 623.848,A -85,B 0,C 180,E1 16475.244,E2 16475.244} C_VEL
LIN {X 0,Y 328.319,Z 625.601,A -85,B 0,C 180,E1 16472.095,E2 16472.095} C_VEL
LIN {X 0,Y 328.345,Z 625.804,A -85,B 0,C 180,E1 16468.954,E2 16468.954} C_VEL
LIN {X 0,Y 328.261,Z 624.468,A -85,B 0,C 180,E1 16465.634,E2 16465.634} C_VEL
LIN {X 0,Y 328.199,Z 621.704,A -85,B 0,C 180,E1 16462.474,E2 16462.474} C_VEL
LIN {X 0,Y 328.311,Z 617.069,A -85,B 0,C 180,E1 16459.117,E2 16459.117} C_VEL
LIN {X 0,Y 328.787,Z 610.702,A -85,B 0,C 180,E1 16455.741,E2 16455.741} C_VEL
LIN {X 0,Y 329.816,Z 602.482,A -85,B 0,C 180,E1 16452.354,E2 16452.354} C_VEL
LIN {X 0,Y 331.417,Z 592.824,A -85,B 0,C 180,E1 16449.147,E2 16449.147} C_VEL
LIN {X 0,Y 333.623,Z 581.585,A -85,B 0,C 180,E1 16446.074,E2 16446.074} C_VEL
LIN {X 0,Y 336.557,Z 568.092,A -85,B 0,C 180,E1 16443.03,E2 16443.03} C_VEL
LIN {X 0,Y 340.021,Z 552.9,A -85,B 0,C 180,E1 16440.202,E2 16440.202} C_VEL
LIN {X 0,Y 343.69,Z 536.892,A -85,B 0,C 180,E1 16437.736,E2 16437.736} C_VEL
LIN {X 0,Y 347.63,Z 519.16,A -85,B 0,C 180,E1 16435.487,E2 16435.487} C_VEL
LIN {X 0,Y 351.565,Z 500.189,A -85,B 0,C 180,E1 16433.532,E2 16433.532} C_VEL
LIN {X 0,Y 355.17,Z 480.898,A -85,B 0,C 180,E1 16431.939,E2 16431.939} C_VEL
LIN {X 0,Y 358.371,Z 461.031,A -85,B 0,C 180,E1 16430.648,E2 16430.648} C_VEL
LIN {X 0,Y 361.062,Z 440.832,A -85,B 0,C 180,E1 16429.656,E2 16429.656} C_VEL
LIN {X 0,Y 363.117,Z 420.347,A -85,B 0,C 180,E1 16428.938,E2 16428.938} C_VEL
LIN {X 0,Y 364.69,Z 390.811,A -85,B 0,C 180,E1 16428.248,E2 16428.248} C_VEL
LIN {X 0,Y 372.849,Z 207.039,A -85,B 0,C 180,E1 16424.393,E2 16424.393} C_VEL
LIN {X 0,Y 362.023,Z 187.503,A -85,B 0,C 180,E1 16422.234,E2 16422.234} C_VEL
LIN {X 0,Y 351.469,Z 170.609,A -85,B 0,C 180,E1 16419.983,E2 16419.983} C_VEL
LIN {X 0,Y 348.203,Z 165.522,A -85,B 0,C 180,E1 16419.177,E2 16419.177} C_VEL
LIN {X 0,Y 343.122,Z 154.359,A -85,B 0,C 180,E1 16416.463,E2 16416.463} C_VEL
LIN {X 0,Y 338.807,Z 145.777,A -85,B 0,C 180,E1 16414.105,E2 16414.105} C_VEL
LIN {X 0,Y 336.724,Z 141.707,A -85,B 0,C 180,E1 16412.915,E2 16412.915} C_VEL
LIN {X 0,Y 334.764,Z 137.713,A -85,B 0,C 180,E1 16411.713,E2 16411.713} C_VEL
LIN {X 0,Y 332.801,Z 134.046,A -85,B 0,C 180,E1 16410.513,E2 16410.513} C_VEL
LIN {X 0,Y 331.924,Z 132.614,A -85,B 0,C 180,E1 16410.002,E2 16410.002} C_VEL
LIN {X 0,Y 330.291,Z 129.705,A -85,B 0,C 180,E1 16408.97,E2 16408.97} C_VEL
LIN {X 0,Y 330.024,Z 128.35,A -85,B 0,C 180,E1 16408.529,E2 16408.529} C_VEL
LIN {X 0,Y 330.031,Z 128.346,A -85,B 0,C 180,E1 16404.233,E2 16404.233} C_VEL
LIN {X 0,Y 330.022,Z 128.353,A -85,B 0,C 180,E1 16400.02,E2 16400.02} C_VEL
LIN {X 0,Y 330.002,Z 128.378,A -85,B 0,C 180,E1 16395.644,E2 16395.644} C_VEL
LIN {X 0,Y 329.994,Z 128.363,A -85,B 0,C 180,E1 16391.358,E2 16391.358} C_VEL
LIN {X 0,Y 329.992,Z 128.342,A -85,B 0,C 180,E1 16387.136,E2 16387.136} C_VEL
LIN {X 0,Y 330.003,Z 128.365,A -85,B 0,C 180,E1 16382.952,E2 16382.952} C_VEL
LIN {X 0,Y 330.023,Z 128.369,A -85,B 0,C 180,E1 16378.611,E2 16378.611} C_VEL
LIN {X 0,Y 330.016,Z 128.339,A -85,B 0,C 180,E1 16374.262,E2 16374.262} C_VEL
LIN {X 0,Y 330.003,Z 128.36,A -85,B 0,C 180,E1 16370.055,E2 16370.055} C_VEL
LIN {X 0,Y 329.993,Z 128.379,A -85,B 0,C 180,E1 16365.793,E2 16365.793} C_VEL
LIN {X 0,Y 329.987,Z 128.35,A -85,B 0,C 180,E1 16361.449,E2 16361.449} C_VEL
LIN {X 0,Y 329.993,Z 128.347,A -85,B 0,C 180,E1 16357.18,E2 16357.18} C_VEL
LIN {X 0,Y 330.007,Z 128.357,A -85,B 0,C 180,E1 16352.966,E2 16352.966} C_VEL
LIN {X 0,Y 330.024,Z 128.367,A -85,B 0,C 180,E1 16348.593,E2 16348.593} C_VEL
LIN {X 0,Y 330.042,Z 128.608,A -85,B 0,C 180,E1 16346.954,E2 16346.954} C_VEL
LIN {X 0,Y 331.585,Z 132.256,A -85,B 0,C 180,E1 16345.71,E2 16345.71} C_VEL
LIN {X 0,Y 332.526,Z 133.619,A -85,B 0,C 180,E1 16345.158,E2 16345.158} C_VEL
LIN {X 0,Y 334.338,Z 137.358,A -85,B 0,C 180,E1 16343.903,E2 16343.903} C_VEL
LIN {X 0,Y 338.789,Z 146.408,A -85,B 0,C 180,E1 16341.051,E2 16341.051} C_VEL
LIN {X 0,Y 344.285,Z 158.82,A -85,B 0,C 180,E1 16337.641,E2 16337.641} C_VEL
LIN {X 0,Y 349.666,Z 172.002,A -85,B 0,C 180,E1 16334.465,E2 16334.465} C_VEL
LIN {X 0,Y 360.068,Z 189.162,A -85,B 0,C 180,E1 16332.236,E2 16332.236} C_VEL
LIN {X 0,Y 368.63,Z 204.931,A -85,B 0,C 180,E1 16330.515,E2 16330.515} C_VEL
LIN {X 0,Y 370.688,Z 220.997,A -85,B 0,C 180,E1 16329.822,E2 16329.822} C_VEL
LIN {X 0,Y 364.531,Z 395.209,A -85,B 0,C 180,E1 16326.507,E2 16326.507} C_VEL
LIN {X 0,Y 363.022,Z 414.636,A -85,B 0,C 180,E1 16325.864,E2 16325.864} C_VEL
LIN {X 0,Y 360.856,Z 433.538,A -85,B 0,C 180,E1 16324.944,E2 16324.944} C_VEL
LIN {X 0,Y 358.099,Z 451.716,A -85,B 0,C 180,E1 16323.753,E2 16323.753} C_VEL
LIN {X 0,Y 354.888,Z 468.936,A -85,B 0,C 180,E1 16322.304,E2 16322.304} C_VEL
LIN {X 0,Y 351.432,Z 484.96,A -85,B 0,C 180,E1 16320.614,E2 16320.614} C_VEL
LIN {X 0,Y 347.678,Z 500.339,A -85,B 0,C 180,E1 16318.607,E2 16318.607} C_VEL
LIN {X 0,Y 344.017,Z 514.121,A -85,B 0,C 180,E1 16316.402,E2 16316.402} C_VEL
LIN {X 0,Y 340.452,Z 526.837,A -85,B 0,C 180,E1 16313.908,E2 16313.908} C_VEL
LIN {X 0,Y 337.214,Z 538.049,A -85,B 0,C 180,E1 16311.206,E2 16311.206} C_VEL
LIN {X 0,Y 334.422,Z 547.79,A -85,B 0,C 180,E1 16308.295,E2 16308.295} C_VEL
LIN {X 0,Y 332.154,Z 556.044,A -85,B 0,C 180,E1 16305.181,E2 16305.181} C_VEL
LIN {X 0,Y 330.464,Z 562.762,A -85,B 0,C 180,E1 16301.872,E2 16301.872} C_VEL
LIN {X 0,Y 329.405,Z 567.659,A -85,B 0,C 180,E1 16298.552,E2 16298.552} C_VEL
LIN {X 0,Y 328.803,Z 570.998,A -85,B 0,C 180,E1 16295.058,E2 16295.058} C_VEL
LIN {X 0,Y 328.569,Z 572.609,A -85,B 0,C 180,E1 16291.568,E2 16291.568} C_VEL
LIN {X 0,Y 328.579,Z 572.551,A -85,B 0,C 180,E1 16288.081,E2 16288.081} C_VEL
LIN {X 0,Y 328.833,Z 570.819,A -85,B 0,C 180,E1 16284.59,E2 16284.59} C_VEL
LIN {X 0,Y 329.429,Z 567.573,A -85,B 0,C 180,E1 16281.27,E2 16281.27} C_VEL
LIN {X 0,Y 330.576,Z 562.315,A -85,B 0,C 180,E1 16277.776,E2 16277.776} C_VEL
LIN {X 0,Y 332.323,Z 555.443,A -85,B 0,C 180,E1 16274.467,E2 16274.467} C_VEL
LIN {X 0,Y 334.618,Z 547.147,A -85,B 0,C 180,E1 16271.391,E2 16271.391} C_VEL
LIN {X 0,Y 334.683,Z 543.68,A -85,B 0,C 180,E1 16270.208,E2 16270.208} C_VEL
LIN {X 0,Y 331.954,Z 534.48,A -85,B 0,C 180,E1 16267.161,E2 16267.161} C_VEL
LIN {X 0,Y 332.352,Z 530.202,A -85,B 0,C 180,E1 16266.044,E2 16266.044} C_VEL
LIN {X 0,Y 335.968,Z 518.033,A -85,B 0,C 180,E1 16263.485,E2 16263.485} C_VEL
LIN {X 0,Y 339.974,Z 503.859,A -85,B 0,C 180,E1 16261.066,E2 16261.066} C_VEL
LIN {X 0,Y 343.976,Z 488.451,A -85,B 0,C 180,E1 16258.938,E2 16258.938} C_VEL
LIN {X 0,Y 347.643,Z 472.599,A -85,B 0,C 180,E1 16257.169,E2 16257.169} C_VEL
LIN {X 0,Y 351.016,Z 455.792,A -85,B 0,C 180,E1 16255.666,E2 16255.666} C_VEL
LIN {X 0,Y 353.976,Z 437.959,A -85,B 0,C 180,E1 16254.416,E2 16254.416} C_VEL
LIN {X 0,Y 356.405,Z 418.872,A -85,B 0,C 180,E1 16253.411,E2 16253.411} C_VEL
LIN {X 0,Y 358.134,Z 399.313,A -85,B 0,C 180,E1 16252.696,E2 16252.696} C_VEL
LIN {X 0,Y 359.291,Z 373.683,A -85,B 0,C 180,E1 16252.131,E2 16252.131} C_VEL
LIN {X 0,Y 364.792,Z 220.41,A -85,B 0,C 180,E1 16249.188,E2 16249.188} C_VEL
LIN {X 0,Y 362.957,Z 208.08,A -85,B 0,C 180,E1 16248.592,E2 16248.592} C_VEL
LIN {X 0,Y 352.342,Z 188.898,A -85,B 0,C 180,E1 16246.355,E2 16246.355} C_VEL
LIN {X 0,Y 341.567,Z 171.531,A -85,B 0,C 180,E1 16243.871,E2 16243.871} C_VEL
LIN {X 0,Y 339.71,Z 166.932,A -85,B 0,C 180,E1 16242.721,E2 16242.721} C_VEL
LIN {X 0,Y 337.217,Z 166.458,A -85,B 0,C 180,E1 16242.091,E2 16242.091} C_VEL
LIN {X 0,Y 344.651,Z 187.706,A -85,B 0,C 180,E1 16238.968,E2 16238.968} C_VEL
LIN {X 0,Y 345.771,Z 190.783,A -85,B 0,C 180,E1 16238.603,E2 16238.603} C_VEL
LIN {X 0,Y 346.447,Z 193.78,A -85,B 0,C 180,E1 16238.436,E2 16238.436} C_VEL
LIN {X 0,Y 348.712,Z 216.697,A -85,B 0,C 180,E1 16237.462,E2 16237.462} C_VEL
LIN {X 0,Y 338.84,Z 402.631,A -85,B 0,C 180,E1 16232.323,E2 16232.323} C_VEL
LIN {X 0,Y 337.503,Z 422.878,A -85,B 0,C 180,E1 16231.427,E2 16231.427} C_VEL
LIN {X 0,Y 335.776,Z 442.731,A -85,B 0,C 180,E1 16230.215,E2 16230.215} C_VEL
LIN {X 0,Y 333.814,Z 461.447,A -85,B 0,C 180,E1 16228.734,E2 16228.734} C_VEL
LIN {X 0,Y 331.705,Z 479.165,A -85,B 0,C 180,E1 16226.979,E2 16226.979} C_VEL
LIN {X 0,Y 329.524,Z 495.749,A -85,B 0,C 180,E1 16224.946,E2 16224.946} C_VEL
LIN {X 0,Y 327.508,Z 510.313,A -85,B 0,C 180,E1 16222.78,E2 16222.78} C_VEL
LIN {X 0,Y 325.583,Z 524.09,A -85,B 0,C 180,E1 16220.306,E2 16220.306} C_VEL
LIN {X 0,Y 323.909,Z 536.464,A -85,B 0,C 180,E1 16217.609,E2 16217.609} C_VEL
LIN {X 0,Y 322.574,Z 547.218,A -85,B 0,C 180,E1 16214.738,E2 16214.738} C_VEL
LIN {X 0,Y 321.629,Z 555.946,A -85,B 0,C 180,E1 16211.84,E2 16211.84} C_VEL
LIN {X 0,Y 321.005,Z 563.166,A -85,B 0,C 180,E1 16208.779,E2 16208.779} C_VEL
LIN {X 0,Y 320.678,Z 568.516,A -85,B 0,C 180,E1 16205.727,E2 16205.727} C_VEL
LIN {X 0,Y 320.58,Z 572.174,A -85,B 0,C 180,E1 16202.682,E2 16202.682} C_VEL
LIN {X 0,Y 320.644,Z 574.234,A -85,B 0,C 180,E1 16199.643,E2 16199.643} C_VEL
LIN {X 0,Y 320.862,Z 574.725,A -85,B 0,C 180,E1 16196.606,E2 16196.606} C_VEL
LIN {X 0,Y 321.347,Z 573.534,A -85,B 0,C 180,E1 16193.39,E2 16193.39} C_VEL
LIN {X 0,Y 322.147,Z 570.792,A -85,B 0,C 180,E1 16190.352,E2 16190.352} C_VEL
LIN {X 0,Y 323.456,Z 566.098,A -85,B 0,C 180,E1 16187.141,E2 16187.141} C_VEL
LIN {X 0,Y 325.214,Z 559.85,A -85,B 0,C 180,E1 16184.12,E2 16184.12} C_VEL
LIN {X 0,Y 327.541,Z 551.778,A -85,B 0,C 180,E1 16181.143,E2 16181.143} C_VEL
LIN {X 0,Y 330.35,Z 542.001,A -85,B 0,C 180,E1 16178.311,E2 16178.311} C_VEL
LIN {X 0,Y 333.676,Z 530.206,A -85,B 0,C 180,E1 16175.574,E2 16175.574} C_VEL
LIN {X 0,Y 337.177,Z 517.232,A -85,B 0,C 180,E1 16173.141,E2 16173.141} C_VEL
LIN {X 0,Y 340.96,Z 502.416,A -85,B 0,C 180,E1 16170.87,E2 16170.87} C_VEL
LIN {X 0,Y 344.853,Z 486.198,A -85,B 0,C 180,E1 16168.833,E2 16168.833} C_VEL
LIN {X 0,Y 348.66,Z 469.146,A -85,B 0,C 180,E1 16167.083,E2 16167.083} C_VEL
LIN {X 0,Y 352.427,Z 450.231,A -85,B 0,C 180,E1 16165.529,E2 16165.529} C_VEL
LIN {X 0,Y 355.923,Z 430.389,A -85,B 0,C 180,E1 16164.246,E2 16164.246} C_VEL
LIN {X 0,Y 358.984,Z 409.911,A -85,B 0,C 180,E1 16163.252,E2 16163.252} C_VEL
LIN {X 0,Y 368.669,Z 351.364,A -85,B 0,C 180,E1 16161.028,E2 16161.028} C_VEL
LIN {X 0,Y 383.823,Z 276.965,A -85,B 0,C 180,E1 16158.286,E2 16158.286} C_VEL
LIN {X 0,Y 389.547,Z 251.759,A -85,B 0,C 180,E1 16157.385,E2 16157.385} C_VEL
LIN {X 0,Y 383.581,Z 273.688,A -85,B 0,C 180,E1 16156.644,E2 16156.644} C_VEL
LIN {X 0,Y 376.965,Z 298.92,A -85,B 0,C 180,E1 16155.752,E2 16155.752} C_VEL
LIN {X 0,Y 370.977,Z 322.986,A -85,B 0,C 180,E1 16154.882,E2 16154.882} C_VEL
LIN {X 0,Y 365.261,Z 347.126,A -85,B 0,C 180,E1 16153.984,E2 16153.984} C_VEL
LIN {X 0,Y 359.865,Z 371.322,A -85,B 0,C 180,E1 16153.062,E2 16153.062} C_VEL
LIN {X 0,Y 359.239,Z 375.828,A -85,B 0,C 180,E1 16152.891,E2 16152.891} C_VEL
LIN {X 0,Y 357.137,Z 417.822,A -85,B 0,C 180,E1 16151.946,E2 16151.946} C_VEL
LIN {X 0,Y 355.065,Z 438.694,A -85,B 0,C 180,E1 16151.232,E2 16151.232} C_VEL
LIN {X 0,Y 352.296,Z 458.992,A -85,B 0,C 180,E1 16150.254,E2 16150.254} C_VEL
LIN {X 0,Y 348.98,Z 478.934,A -85,B 0,C 180,E1 16148.969,E2 16148.969} C_VEL
LIN {X 0,Y 345.384,Z 497.545,A -85,B 0,C 180,E1 16147.441,E2 16147.441} C_VEL
LIN {X 0,Y 341.543,Z 515.383,A -85,B 0,C 180,E1 16145.632,E2 16145.632} C_VEL
LIN {X 0,Y 337.619,Z 532.393,A -85,B 0,C 180,E1 16143.527,E2 16143.527} C_VEL
LIN {X 0,Y 333.748,Z 548.484,A -85,B 0,C 180,E1 16141.118,E2 16141.118} C_VEL
LIN {X 0,Y 330.095,Z 563.544,A -85,B 0,C 180,E1 16138.396,E2 16138.396} C_VEL
LIN {X 0,Y 327.011,Z 576.699,A -85,B 0,C 180,E1 16135.54,E2 16135.54} C_VEL
LIN {X 0,Y 324.443,Z 588.486,A -85,B 0,C 180,E1 16132.467,E2 16132.467} C_VEL
LIN {X 0,Y 322.479,Z 598.856,A -85,B 0,C 180,E1 16129.188,E2 16129.188} C_VEL
LIN {X 0,Y 321.147,Z 607.687,A -85,B 0,C 180,E1 16125.717,E2 16125.717} C_VEL
LIN {X 0,Y 320.445,Z 614.596,A -85,B 0,C 180,E1 16122.251,E2 16122.251} C_VEL
LIN {X 0,Y 320.22,Z 619.737,A -85,B 0,C 180,E1 16118.802,E2 16118.802} C_VEL
LIN {X 0,Y 320.255,Z 623.198,A -85,B 0,C 180,E1 16115.375,E2 16115.375} C_VEL
LIN {X 0,Y 320.342,Z 624.955,A -85,B 0,C 180,E1 16112.148,E2 16112.148} C_VEL
LIN {X 0,Y 320.37,Z 625.159,A -85,B 0,C 180,E1 16108.928,E2 16108.928} C_VEL
LIN {X 0,Y 320.283,Z 623.943,A -85,B 0,C 180,E1 16105.704,E2 16105.704} C_VEL
LIN {X 0,Y 320.213,Z 621.225,A -85,B 0,C 180,E1 16102.465,E2 16102.465} C_VEL
LIN {X 0,Y 320.308,Z 616.957,A -85,B 0,C 180,E1 16099.206,E2 16099.206} C_VEL
LIN {X 0,Y 320.82,Z 610.404,A -85,B 0,C 180,E1 16095.564,E2 16095.564} C_VEL
LIN {X 0,Y 321.903,Z 602.279,A -85,B 0,C 180,E1 16092.093,E2 16092.093} C_VEL
LIN {X 0,Y 323.592,Z 592.723,A -85,B 0,C 180,E1 16088.808,E2 16088.808} C_VEL
LIN {X 0,Y 326.016,Z 581.096,A -85,B 0,C 180,E1 16085.543,E2 16085.543} C_VEL
LIN {X 0,Y 329.057,Z 567.911,A -85,B 0,C 180,E1 16082.494,E2 16082.494} C_VEL
LIN {X 0,Y 332.734,Z 552.678,A -85,B 0,C 180,E1 16079.59,E2 16079.59} C_VEL
LIN {X 0,Y 336.592,Z 536.665,A -85,B 0,C 180,E1 16077.072,E2 16077.072} C_VEL
LIN {X 0,Y 340.549,Z 519.682,A -85,B 0,C 180,E1 16074.87,E2 16074.87} C_VEL
LIN {X 0,Y 344.275,Z 502.592,A -85,B 0,C 180,E1 16073.047,E2 16073.047} C_VEL
LIN {X 0,Y 347.984,Z 483.956,A -85,B 0,C 180,E1 16071.429,E2 16071.429} C_VEL
LIN {X 0,Y 351.373,Z 464.435,A -85,B 0,C 180,E1 16070.085,E2 16070.085} C_VEL
LIN {X 0,Y 354.338,Z 443.765,A -85,B 0,C 180,E1 16069,E2 16069} C_VEL
LIN {X 0,Y 356.655,Z 422.759,A -85,B 0,C 180,E1 16068.215,E2 16068.215} C_VEL
LIN {X 0,Y 358.131,Z 399.138,A -85,B 0,C 180,E1 16067.62,E2 16067.62} C_VEL
LIN {X 0,Y 366.817,Z 210.027,A -85,B 0,C 180,E1 16063.6,E2 16063.6} C_VEL
LIN {X 0,Y 356.836,Z 192.006,A -85,B 0,C 180,E1 16061.531,E2 16061.531} C_VEL
LIN {X 0,Y 347.107,Z 176.238,A -85,B 0,C 180,E1 16059.378,E2 16059.378} C_VEL
LIN {X 0,Y 340.396,Z 166.061,A -85,B 0,C 180,E1 16057.765,E2 16057.765} C_VEL
LIN {X 0,Y 334.989,Z 154.611,A -85,B 0,C 180,E1 16054.756,E2 16054.756} C_VEL
LIN {X 0,Y 331.148,Z 147.066,A -85,B 0,C 180,E1 16052.51,E2 16052.51} C_VEL
LIN {X 0,Y 329.189,Z 143.175,A -85,B 0,C 180,E1 16051.291,E2 16051.291} C_VEL
LIN {X 0,Y 327.035,Z 138.913,A -85,B 0,C 180,E1 16049.89,E2 16049.89} C_VEL
LIN {X 0,Y 325.112,Z 135.585,A -85,B 0,C 180,E1 16048.67,E2 16048.67} C_VEL
LIN {X 0,Y 324.411,Z 134.036,A -85,B 0,C 180,E1 16048.135,E2 16048.135} C_VEL
LIN {X 0,Y 322.498,Z 131.131,A -85,B 0,C 180,E1 16046.914,E2 16046.914} C_VEL
LIN {X 0,Y 322.093,Z 129.366,A -85,B 0,C 180,E1 16046.353,E2 16046.353} C_VEL
LIN {X 0,Y 322.09,Z 129.355,A -85,B 0,C 180,E1 16042.062,E2 16042.062} C_VEL
LIN {X 0,Y 322.062,Z 129.342,A -85,B 0,C 180,E1 16037.622,E2 16037.622} C_VEL
LIN {X 0,Y 322.055,Z 129.332,A -85,B 0,C 180,E1 16033.282,E2 16033.282} C_VEL
LIN {X 0,Y 322.064,Z 129.348,A -85,B 0,C 180,E1 16028.93,E2 16028.93} C_VEL
LIN {X 0,Y 322.081,Z 129.362,A -85,B 0,C 180,E1 16024.629,E2 16024.629} C_VEL
LIN {X 0,Y 322.077,Z 129.329,A -85,B 0,C 180,E1 16020.178,E2 16020.178} C_VEL
LIN {X 0,Y 322.057,Z 129.339,A -85,B 0,C 180,E1 16015.905,E2 16015.905} C_VEL
LIN {X 0,Y 322.054,Z 129.37,A -85,B 0,C 180,E1 16011.609,E2 16011.609} C_VEL
LIN {X 0,Y 322.06,Z 129.34,A -85,B 0,C 180,E1 16007.083,E2 16007.083} C_VEL
LIN {X 0,Y 322.069,Z 129.332,A -85,B 0,C 180,E1 16002.846,E2 16002.846} C_VEL
LIN {X 0,Y 322.088,Z 129.349,A -85,B 0,C 180,E1 15998.511,E2 15998.511} C_VEL
LIN {X 0,Y 322.059,Z 129.366,A -85,B 0,C 180,E1 15994.039,E2 15994.039} C_VEL
LIN {X 0,Y 322.046,Z 129.36,A -85,B 0,C 180,E1 15989.597,E2 15989.597} C_VEL
LIN {X 0,Y 322.077,Z 129.503,A -85,B 0,C 180,E1 15989.187,E2 15989.187} C_VEL
LIN {X 0,Y 323.547,Z 133.106,A -85,B 0,C 180,E1 15987.856,E2 15987.856} C_VEL
LIN {X 0,Y 324.67,Z 134.565,A -85,B 0,C 180,E1 15987.179,E2 15987.179} C_VEL
LIN {X 0,Y 326.531,Z 138.467,A -85,B 0,C 180,E1 15985.764,E2 15985.764} C_VEL
LIN {X 0,Y 329.806,Z 145.196,A -85,B 0,C 180,E1 15983.453,E2 15983.453} C_VEL
LIN {X 0,Y 333.544,Z 153.07,A -85,B 0,C 180,E1 15980.985,E2 15980.985} C_VEL
LIN {X 0,Y 338.199,Z 163.399,A -85,B 0,C 180,E1 15978.075,E2 15978.075} C_VEL
LIN {X 0,Y 341.901,Z 172.256,A -85,B 0,C 180,E1 15975.892,E2 15975.892} C_VEL
LIN {X 0,Y 352.617,Z 189.518,A -85,B 0,C 180,E1 15973.456,E2 15973.456} C_VEL
LIN {X 0,Y 362.859,Z 208.049,A -85,B 0,C 180,E1 15971.303,E2 15971.303} C_VEL
LIN {X 0,Y 364.816,Z 221.552,A -85,B 0,C 180,E1 15970.665,E2 15970.665} C_VEL
LIN {X 0,Y 358.342,Z 395.462,A -85,B 0,C 180,E1 15967.31,E2 15967.31} C_VEL
LIN {X 0,Y 356.775,Z 414.874,A -85,B 0,C 180,E1 15966.661,E2 15966.661} C_VEL
LIN {X 0,Y 354.59,Z 433.343,A -85,B 0,C 180,E1 15965.759,E2 15965.759} C_VEL
LIN {X 0,Y 351.713,Z 451.704,A -85,B 0,C 180,E1 15964.55,E2 15964.55} C_VEL
LIN {X 0,Y 348.3,Z 469.318,A -85,B 0,C 180,E1 15963.053,E2 15963.053} C_VEL
LIN {X 0,Y 344.597,Z 485.765,A -85,B 0,C 180,E1 15961.289,E2 15961.289} C_VEL
LIN {X 0,Y 340.687,Z 501.096,A -85,B 0,C 180,E1 15959.25,E2 15959.25} C_VEL
LIN {X 0,Y 336.871,Z 514.844,A -85,B 0,C 180,E1 15957.007,E2 15957.007} C_VEL
LIN {X 0,Y 333.141,Z 527.536,A -85,B 0,C 180,E1 15954.466,E2 15954.466} C_VEL
LIN {X 0,Y 329.746,Z 538.732,A -85,B 0,C 180,E1 15951.71,E2 15951.71} C_VEL
LIN {X 0,Y 326.809,Z 548.462,A -85,B 0,C 180,E1 15948.737,E2 15948.737} C_VEL
LIN {X 0,Y 324.415,Z 556.706,A -85,B 0,C 180,E1 15945.552,E2 15945.552} C_VEL
LIN {X 0,Y 322.621,Z 563.416,A -85,B 0,C 180,E1 15942.165,E2 15942.165} C_VEL
LIN {X 0,Y 321.492,Z 568.31,A -85,B 0,C 180,E1 15938.764,E2 15938.764} C_VEL
LIN {X 0,Y 320.847,Z 571.645,A -85,B 0,C 180,E1 15935.184,E2 15935.184} C_VEL
LIN {X 0,Y 320.597,Z 573.254,A -85,B 0,C 180,E1 15931.607,E2 15931.607} C_VEL
LIN {X 0,Y 320.607,Z 573.196,A -85,B 0,C 180,E1 15928.033,E2 15928.033} C_VEL
LIN {X 0,Y 320.88,Z 571.467,A -85,B 0,C 180,E1 15924.456,E2 15924.456} C_VEL
LIN {X 0,Y 321.563,Z 567.99,A -85,B 0,C 180,E1 15920.875,E2 15920.875} C_VEL
LIN {X 0,Y 322.742,Z 562.972,A -85,B 0,C 180,E1 15917.474,E2 15917.474} C_VEL
LIN {X 0,Y 324.596,Z 556.107,A -85,B 0,C 180,E1 15914.088,E2 15914.088} C_VEL
LIN {X 0,Y 327.051,Z 547.706,A -85,B 0,C 180,E1 15910.905,E2 15910.905} C_VEL
LIN {X 0,Y 330.051,Z 537.805,A -85,B 0,C 180,E1 15907.935,E2 15907.935} C_VEL
LIN {X 0,Y 332.352,Z 530.202,A -85,B 0,C 180,E1 15906.044,E2 15906.044} C_VEL
LIN {X 0,Y 332.815,Z 525.768,A -85,B 0,C 180,E1 15904.953,E2 15904.953} C_VEL
LIN {X 0,Y 331.018,Z 514.323,A -85,B 0,C 180,E1 15902.12,E2 15902.12} C_VEL
LIN {X 0,Y 331.72,Z 509.097,A -85,B 0,C 180,E1 15901.121,E2 15901.121} C_VEL
LIN {X 0,Y 335.688,Z 494.932,A -85,B 0,C 180,E1 15898.982,E2 15898.982} C_VEL
LIN {X 0,Y 339.569,Z 479.583,A -85,B 0,C 180,E1 15897.093,E2 15897.093} C_VEL
LIN {X 0,Y 343.179,Z 463.34,A -85,B 0,C 180,E1 15895.48,E2 15895.48} C_VEL
LIN {X 0,Y 346.396,Z 446.231,A -85,B 0,C 180,E1 15894.129,E2 15894.129} C_VEL
LIN {X 0,Y 349.118,Z 428.15,A -85,B 0,C 180,E1 15893.027,E2 15893.027} C_VEL
LIN {X 0,Y 351.245,Z 409.073,A -85,B 0,C 180,E1 15892.179,E2 15892.179} C_VEL
LIN {X 0,Y 352.602,Z 389.477,A -85,B 0,C 180,E1 15891.606,E2 15891.606} C_VEL
LIN {X 0,Y 358.988,Z 221.843,A -85,B 0,C 180,E1 15888.336,E2 15888.336} C_VEL
LIN {X 0,Y 357.556,Z 212.077,A -85,B 0,C 180,E1 15887.85,E2 15887.85} C_VEL
LIN {X 0,Y 347.797,Z 194.224,A -85,B 0,C 180,E1 15885.712,E2 15885.712} C_VEL
LIN {X 0,Y 337.341,Z 177.25,A -85,B 0,C 180,E1 15883.239,E2 15883.239} C_VEL
LIN {X 0,Y 334.971,Z 173.926,A -85,B 0,C 180,E1 15882.655,E2 15882.655} C_VEL
LIN {X 0,Y 333.03,Z 174.235,A -85,B 0,C 180,E1 15882.262,E2 15882.262} C_VEL
LIN {X 0,Y 331.76,Z 173.712,A -85,B 0,C 180,E1 15881.931,E2 15881.931} C_VEL
LIN {X 0,Y 337.805,Z 190.978,A -85,B 0,C 180,E1 15879.417,E2 15879.417} C_VEL
LIN {X 0,Y 339.644,Z 195.685,A -85,B 0,C 180,E1 15879.064,E2 15879.064} C_VEL
LIN {X 0,Y 341.722,Z 217.839,A -85,B 0,C 180,E1 15878.097,E2 15878.097} C_VEL
LIN {X 0,Y 331.421,Z 403.323,A -85,B 0,C 180,E1 15872.827,E2 15872.827} C_VEL
LIN {X 0,Y 330.041,Z 423.429,A -85,B 0,C 180,E1 15871.915,E2 15871.915} C_VEL
LIN {X 0,Y 328.281,Z 443.002,A -85,B 0,C 180,E1 15870.696,E2 15870.696} C_VEL
LIN {X 0,Y 326.227,Z 461.984,A -85,B 0,C 180,E1 15869.165,E2 15869.165} C_VEL
LIN {X 0,Y 324.047,Z 479.725,A -85,B 0,C 180,E1 15867.371,E2 15867.371} C_VEL
LIN {X 0,Y 321.78,Z 496.428,A -85,B 0,C 180,E1 15865.28,E2 15865.28} C_VEL
LIN {X 0,Y 319.657,Z 511.296,A -85,B 0,C 180,E1 15863.016,E2 15863.016} C_VEL
LIN {X 0,Y 317.655,Z 525.212,A -85,B 0,C 180,E1 15860.45,E2 15860.45} C_VEL
LIN {X 0,Y 315.942,Z 537.523,A -85,B 0,C 180,E1 15857.687,E2 15857.687} C_VEL
LIN {X 0,Y 314.645,Z 547.639,A -85,B 0,C 180,E1 15854.916,E2 15854.916} C_VEL
LIN {X 0,Y 313.639,Z 556.713,A -85,B 0,C 180,E1 15851.844,E2 15851.844} C_VEL
LIN {X 0,Y 313.024,Z 563.698,A -85,B 0,C 180,E1 15848.82,E2 15848.82} C_VEL
LIN {X 0,Y 312.692,Z 569.128,A -85,B 0,C 180,E1 15845.689,E2 15845.689} C_VEL
LIN {X 0,Y 312.6,Z 572.851,A -85,B 0,C 180,E1 15842.567,E2 15842.567} C_VEL
LIN {X 0,Y 312.68,Z 574.963,A -85,B 0,C 180,E1 15839.451,E2 15839.451} C_VEL
LIN {X 0,Y 312.957,Z 575.478,A -85,B 0,C 180,E1 15836.153,E2 15836.153} C_VEL
LIN {X 0,Y 313.48,Z 574.368,A -85,B 0,C 180,E1 15833.039,E2 15833.039} C_VEL
LIN {X 0,Y 314.44,Z 571.477,A -85,B 0,C 180,E1 15829.743,E2 15829.743} C_VEL
LIN {X 0,Y 315.828,Z 567.055,A -85,B 0,C 180,E1 15826.638,E2 15826.638} C_VEL
LIN {X 0,Y 317.773,Z 560.924,A -85,B 0,C 180,E1 15823.55,E2 15823.55} C_VEL
LIN {X 0,Y 320.5,Z 552.344,A -85,B 0,C 180,E1 15820.311,E2 15820.311} C_VEL
LIN {X 0,Y 323.756,Z 542.044,A -85,B 0,C 180,E1 15817.292,E2 15817.292} C_VEL
LIN {X 0,Y 327.198,Z 530.869,A -85,B 0,C 180,E1 15814.671,E2 15814.671} C_VEL
LIN {X 0,Y 331.187,Z 517.352,A -85,B 0,C 180,E1 15812.099,E2 15812.099} C_VEL
LIN {X 0,Y 335.437,Z 502.211,A -85,B 0,C 180,E1 15809.752,E2 15809.752} C_VEL
LIN {X 0,Y 339.888,Z 485.436,A -85,B 0,C 180,E1 15807.63,E2 15807.63} C_VEL
LIN {X 0,Y 344.422,Z 466.571,A -85,B 0,C 180,E1 15805.724,E2 15805.724} C_VEL
LIN {X 0,Y 348.611,Z 447.649,A -85,B 0,C 180,E1 15804.191,E2 15804.191} C_VEL
LIN {X 0,Y 352.615,Z 426.626,A -85,B 0,C 180,E1 15802.884,E2 15802.884} C_VEL
LIN {X 0,Y 356.408,Z 403.596,A -85,B 0,C 180,E1 15801.826,E2 15801.826} C_VEL
LIN {X 0,Y 368.709,Z 339.552,A -85,B 0,C 180,E1 15799.371,E2 15799.371} C_VEL
LIN {X 0,Y 380.389,Z 287.45,A -85,B 0,C 180,E1 15797.434,E2 15797.434} C_VEL
LIN {X 0,Y 374.793,Z 307.593,A -85,B 0,C 180,E1 15796.717,E2 15796.717} C_VEL
LIN {X 0,Y 368.154,Z 332.489,A -85,B 0,C 180,E1 15795.821,E2 15795.821} C_VEL
LIN {X 0,Y 362.091,Z 356.409,A -85,B 0,C 180,E1 15794.929,E2 15794.929} C_VEL
LIN {X 0,Y 357.582,Z 375.235,A -85,B 0,C 180,E1 15794.17,E2 15794.17} C_VEL
LIN {X 0,Y 353.046,Z 394.885,A -85,B 0,C 180,E1 15793.447,E2 15793.447} C_VEL
LIN {X 0,Y 351.975,Z 401.173,A -85,B 0,C 180,E1 15793.182,E2 15793.182} C_VEL
LIN {X 0,Y 350.477,Z 423.339,A -85,B 0,C 180,E1 15792.604,E2 15792.604} C_VEL
LIN {X 0,Y 348.082,Z 444.019,A -85,B 0,C 180,E1 15791.814,E2 15791.814} C_VEL
LIN {X 0,Y 345.098,Z 463.955,A -85,B 0,C 180,E1 15790.755,E2 15790.755} C_VEL
LIN {X 0,Y 341.449,Z 484.128,A -85,B 0,C 180,E1 15789.345,E2 15789.345} C_VEL
LIN {X 0,Y 337.4,Z 503.467,A -85,B 0,C 180,E1 15787.624,E2 15787.624} C_VEL
LIN {X 0,Y 333.123,Z 521.957,A -85,B 0,C 180,E1 15785.571,E2 15785.571} C_VEL
LIN {X 0,Y 329.022,Z 538.573,A -85,B 0,C 180,E1 15783.313,E2 15783.313} C_VEL
LIN {X 0,Y 325.105,Z 553.961,A -85,B 0,C 180,E1 15780.786,E2 15780.786} C_VEL
LIN {X 0,Y 321.458,Z 568.289,A -85,B 0,C 180,E1 15777.952,E2 15777.952} C_VEL
LIN {X 0,Y 318.333,Z 581.125,A -85,B 0,C 180,E1 15774.892,E2 15774.892} C_VEL
LIN {X 0,Y 315.783,Z 592.657,A -85,B 0,C 180,E1 15771.55,E2 15771.55} C_VEL
LIN {X 0,Y 313.923,Z 602.592,A -85,B 0,C 180,E1 15767.997,E2 15767.997} C_VEL
LIN {X 0,Y 312.814,Z 610.503,A -85,B 0,C 180,E1 15764.438,E2 15764.438} C_VEL
LIN {X 0,Y 312.317,Z 616.579,A -85,B 0,C 180,E1 15760.889,E2 15760.889} C_VEL
LIN {X 0,Y 312.226,Z 620.932,A -85,B 0,C 180,E1 15757.361,E2 15757.361} C_VEL
LIN {X 0,Y 312.31,Z 623.544,A -85,B 0,C 180,E1 15754.04,E2 15754.04} C_VEL
LIN {X 0,Y 312.397,Z 624.565,A -85,B 0,C 180,E1 15750.735,E2 15750.735} C_VEL
LIN {X 0,Y 312.36,Z 624.156,A -85,B 0,C 180,E1 15747.433,E2 15747.433} C_VEL
LIN {X 0,Y 312.253,Z 622.287,A -85,B 0,C 180,E1 15744.12,E2 15744.12} C_VEL
LIN {X 0,Y 312.242,Z 618.843,A -85,B 0,C 180,E1 15740.788,E2 15740.788} C_VEL
LIN {X 0,Y 312.51,Z 613.586,A -85,B 0,C 180,E1 15737.247,E2 15737.247} C_VEL
LIN {X 0,Y 313.313,Z 606.551,A -85,B 0,C 180,E1 15733.692,E2 15733.692} C_VEL
LIN {X 0,Y 314.695,Z 598.134,A -85,B 0,C 180,E1 15730.32,E2 15730.32} C_VEL
LIN {X 0,Y 316.95,Z 587.132,A -85,B 0,C 180,E1 15726.777,E2 15726.777} C_VEL
LIN {X 0,Y 319.921,Z 574.451,A -85,B 0,C 180,E1 15723.455,E2 15723.455} C_VEL
LIN {X 0,Y 323.521,Z 560.081,A -85,B 0,C 180,E1 15720.366,E2 15720.366} C_VEL
LIN {X 0,Y 327.525,Z 544.467,A -85,B 0,C 180,E1 15717.606,E2 15717.606} C_VEL
LIN {X 0,Y 331.698,Z 527.705,A -85,B 0,C 180,E1 15715.166,E2 15715.166} C_VEL
LIN {X 0,Y 335.77,Z 510.615,A -85,B 0,C 180,E1 15713.13,E2 15713.13} C_VEL
LIN {X 0,Y 339.65,Z 492.756,A -85,B 0,C 180,E1 15711.387,E2 15711.387} C_VEL
LIN {X 0,Y 343.254,Z 474.218,A -85,B 0,C 180,E1 15709.93,E2 15709.93} C_VEL
LIN {X 0,Y 346.563,Z 454.384,A -85,B 0,C 180,E1 15708.712,E2 15708.712} C_VEL
LIN {X 0,Y 349.264,Z 434.273,A -85,B 0,C 180,E1 15707.791,E2 15707.791} C_VEL
LIN {X 0,Y 351.21,Z 413.649,A -85,B 0,C 180,E1 15707.126,E2 15707.126} C_VEL
LIN {X 0,Y 360.96,Z 213.393,A -85,B 0,C 180,E1 15702.806,E2 15702.806} C_VEL
LIN {X 0,Y 352.23,Z 197.357,A -85,B 0,C 180,E1 15700.921,E2 15700.921} C_VEL
LIN {X 0,Y 342.712,Z 181.762,A -85,B 0,C 180,E1 15698.741,E2 15698.741} C_VEL
LIN {X 0,Y 332.383,Z 166.152,A -85,B 0,C 180,E1 15696.128,E2 15696.128} C_VEL
LIN {X 0,Y 326.497,Z 153.904,A -85,B 0,C 180,E1 15692.614,E2 15692.614} C_VEL
LIN {X 0,Y 323.492,Z 148.343,A -85,B 0,C 180,E1 15690.77,E2 15690.77} C_VEL
LIN {X 0,Y 321.504,Z 144.415,A -85,B 0,C 180,E1 15689.43,E2 15689.43} C_VEL
LIN {X 0,Y 319.211,Z 140.002,A -85,B 0,C 180,E1 15687.821,E2 15687.821} C_VEL
LIN {X 0,Y 317.205,Z 136.419,A -85,B 0,C 180,E1 15686.387,E2 15686.387} C_VEL
LIN {X 0,Y 316.496,Z 135.088,A -85,B 0,C 180,E1 15685.846,E2 15685.846} C_VEL
LIN {X 0,Y 314.535,Z 131.976,A -85,B 0,C 180,E1 15684.409,E2 15684.409} C_VEL
LIN {X 0,Y 314.134,Z 130.324,A -85,B 0,C 180,E1 15683.842,E2 15683.842} C_VEL
LIN {X 0,Y 314.123,Z 130.325,A -85,B 0,C 180,E1 15679.525,E2 15679.525} C_VEL
LIN {X 0,Y 314.12,Z 130.343,A -85,B 0,C 180,E1 15675.13,E2 15675.13} C_VEL
LIN {X 0,Y 314.14,Z 130.352,A -85,B 0,C 180,E1 15670.638,E2 15670.638} C_VEL
LIN {X 0,Y 314.144,Z 130.319,A -85,B 0,C 180,E1 15666.212,E2 15666.212} C_VEL
LIN {X 0,Y 314.12,Z 130.321,A -85,B 0,C 180,E1 15661.824,E2 15661.824} C_VEL
LIN {X 0,Y 314.117,Z 130.355,A -85,B 0,C 180,E1 15657.263,E2 15657.263} C_VEL
LIN {X 0,Y 314.128,Z 130.333,A -85,B 0,C 180,E1 15652.869,E2 15652.869} C_VEL
LIN {X 0,Y 314.137,Z 130.316,A -85,B 0,C 180,E1 15648.432,E2 15648.432} C_VEL
LIN {X 0,Y 314.119,Z 130.335,A -85,B 0,C 180,E1 15643.999,E2 15643.999} C_VEL
LIN {X 0,Y 314.113,Z 130.358,A -85,B 0,C 180,E1 15639.504,E2 15639.504} C_VEL
LIN {X 0,Y 314.12,Z 130.336,A -85,B 0,C 180,E1 15635.113,E2 15635.113} C_VEL
LIN {X 0,Y 314.134,Z 130.517,A -85,B 0,C 180,E1 15631.689,E2 15631.689} C_VEL
LIN {X 0,Y 315.662,Z 134.153,A -85,B 0,C 180,E1 15630.178,E2 15630.178} C_VEL
LIN {X 0,Y 316.942,Z 136.016,A -85,B 0,C 180,E1 15629.265,E2 15629.265} C_VEL
LIN {X 0,Y 318.786,Z 139.656,A -85,B 0,C 180,E1 15627.778,E2 15627.778} C_VEL
LIN {X 0,Y 321.983,Z 146.057,A -85,B 0,C 180,E1 15625.37,E2 15625.37} C_VEL
LIN {X 0,Y 325.702,Z 153.545,A -85,B 0,C 180,E1 15622.788,E2 15622.788} C_VEL
LIN {X 0,Y 330.963,Z 165.297,A -85,B 0,C 180,E1 15619.266,E2 15619.266} C_VEL
LIN {X 0,Y 333.889,Z 172.066,A -85,B 0,C 180,E1 15617.495,E2 15617.495} C_VEL
LIN {X 0,Y 345.012,Z 189.687,A -85,B 0,C 180,E1 15614.792,E2 15614.792} C_VEL
LIN {X 0,Y 354.704,Z 206.831,A -85,B 0,C 180,E1 15612.631,E2 15612.631} C_VEL
LIN {X 0,Y 357.755,Z 212.914,A -85,B 0,C 180,E1 15611.976,E2 15611.976} C_VEL
LIN {X 0,Y 358.956,Z 223.848,A -85,B 0,C 180,E1 15611.501,E2 15611.501} C_VEL
LIN {X 0,Y 352.22,Z 395.769,A -85,B 0,C 180,E1 15608.14,E2 15608.14} C_VEL
LIN {X 0,Y 350.587,Z 415.216,A -85,B 0,C 180,E1 15607.482,E2 15607.482} C_VEL
LIN {X 0,Y 348.289,Z 433.849,A -85,B 0,C 180,E1 15606.56,E2 15606.56} C_VEL
LIN {X 0,Y 345.397,Z 451.682,A -85,B 0,C 180,E1 15605.376,E2 15605.376} C_VEL
LIN {X 0,Y 341.846,Z 469.395,A -85,B 0,C 180,E1 15603.86,E2 15603.86} C_VEL
LIN {X 0,Y 337.984,Z 485.917,A -85,B 0,C 180,E1 15602.073,E2 15602.073} C_VEL
LIN {X 0,Y 333.899,Z 501.312,A -85,B 0,C 180,E1 15600.004,E2 15600.004} C_VEL
LIN {X 0,Y 329.763,Z 515.565,A -85,B 0,C 180,E1 15597.638,E2 15597.638} C_VEL
LIN {X 0,Y 325.865,Z 528.233,A -85,B 0,C 180,E1 15595.05,E2 15595.05} C_VEL
LIN {X 0,Y 322.305,Z 539.413,A -85,B 0,C 180,E1 15592.238,E2 15592.238} C_VEL
LIN {X 0,Y 319.216,Z 549.132,A -85,B 0,C 180,E1 15589.2,E2 15589.2} C_VEL
LIN {X 0,Y 316.691,Z 557.367,A -85,B 0,C 180,E1 15585.941,E2 15585.941} C_VEL
LIN {X 0,Y 314.786,Z 564.07,A -85,B 0,C 180,E1 15582.472,E2 15582.472} C_VEL
LIN {X 0,Y 313.583,Z 568.96,A -85,B 0,C 180,E1 15578.987,E2 15578.987} C_VEL
LIN {X 0,Y 312.892,Z 572.292,A -85,B 0,C 180,E1 15575.316,E2 15575.316} C_VEL
LIN {X 0,Y 312.625,Z 573.899,A -85,B 0,C 180,E1 15571.648,E2 15571.648} C_VEL
LIN {X 0,Y 312.636,Z 573.842,A -85,B 0,C 180,E1 15567.983,E2 15567.983} C_VEL
LIN {X 0,Y 312.928,Z 572.114,A -85,B 0,C 180,E1 15564.314,E2 15564.314} C_VEL
LIN {X 0,Y 313.66,Z 568.642,A -85,B 0,C 180,E1 15560.643,E2 15560.643} C_VEL
LIN {X 0,Y 314.964,Z 563.442,A -85,B 0,C 180,E1 15557.055,E2 15557.055} C_VEL
LIN {X 0,Y 316.884,Z 556.769,A -85,B 0,C 180,E1 15553.69,E2 15553.69} C_VEL
LIN {X 0,Y 319.533,Z 548.181,A -85,B 0,C 180,E1 15550.369,E2 15550.369} C_VEL
LIN {X 0,Y 322.629,Z 538.491,A -85,B 0,C 180,E1 15547.399,E2 15547.399} C_VEL
LIN {X 0,Y 326.254,Z 527.121,A -85,B 0,C 180,E1 15544.591,E2 15544.591} C_VEL
LIN {X 0,Y 330.215,Z 514.224,A -85,B 0,C 180,E1 15542.008,E2 15542.008} C_VEL
LIN {X 0,Y 331.72,Z 509.097,A -85,B 0,C 180,E1 15541.121,E2 15541.121} C_VEL
LIN {X 0,Y 332.478,Z 503.798,A -85,B 0,C 180,E1 15540.149,E2 15540.149} C_VEL
LIN {X 0,Y 331.294,Z 490.944,A -85,B 0,C 180,E1 15537.738,E2 15537.738} C_VEL
LIN {X 0,Y 331.786,Z 485.004,A -85,B 0,C 180,E1 15536.881,E2 15536.881} C_VEL
LIN {X 0,Y 331.986,Z 484.102,A -85,B 0,C 180,E1 15536.774,E2 15536.774} C_VEL
LIN {X 0,Y 335.895,Z 467.789,A -85,B 0,C 180,E1 15535.038,E2 15535.038} C_VEL
LIN {X 0,Y 339.409,Z 450.619,A -85,B 0,C 180,E1 15533.586,E2 15533.586} C_VEL
LIN {X 0,Y 342.323,Z 433.088,A -85,B 0,C 180,E1 15532.43,E2 15532.43} C_VEL
LIN {X 0,Y 344.722,Z 414.003,A -85,B 0,C 180,E1 15531.499,E2 15531.499} C_VEL
LIN {X 0,Y 346.341,Z 394.6,A -85,B 0,C 180,E1 15530.857,E2 15530.857} C_VEL
LIN {X 0,Y 353.254,Z 223.149,A -85,B 0,C 180,E1 15527.45,E2 15527.45} C_VEL
LIN {X 0,Y 352.226,Z 216.048,A -85,B 0,C 180,E1 15527.087,E2 15527.087} C_VEL
LIN {X 0,Y 342.704,Z 198.566,A -85,B 0,C 180,E1 15524.915,E2 15524.915} C_VEL
LIN {X 0,Y 333.222,Z 182.966,A -85,B 0,C 180,E1 15522.581,E2 15522.581} C_VEL
LIN {X 0,Y 332.63,Z 182.421,A -85,B 0,C 180,E1 15522.441,E2 15522.441} C_VEL
LIN {X 0,Y 329.922,Z 184.332,A -85,B 0,C 180,E1 15521.932,E2 15521.932} C_VEL
LIN {X 0,Y 327.739,Z 184.147,A -85,B 0,C 180,E1 15521.455,E2 15521.455} C_VEL
LIN {X 0,Y 327.304,Z 183.829,A -85,B 0,C 180,E1 15521.341,E2 15521.341} C_VEL
LIN {X 0,Y 330.012,Z 191.587,A -85,B 0,C 180,E1 15520.225,E2 15520.225} C_VEL
LIN {X 0,Y 332.945,Z 198.567,A -85,B 0,C 180,E1 15519.661,E2 15519.661} C_VEL
LIN {X 0,Y 334.759,Z 218.859,A -85,B 0,C 180,E1 15518.756,E2 15518.756} C_VEL
LIN {X 0,Y 324.044,Z 403.455,A -85,B 0,C 180,E1 15513.368,E2 15513.368} C_VEL
LIN {X 0,Y 322.597,Z 423.774,A -85,B 0,C 180,E1 15512.426,E2 15512.426} C_VEL
LIN {X 0,Y 320.749,Z 443.575,A -85,B 0,C 180,E1 15511.163,E2 15511.163} C_VEL
LIN {X 0,Y 318.651,Z 462.313,A -85,B 0,C 180,E1 15509.618,E2 15509.618} C_VEL
LIN {X 0,Y 316.362,Z 480.352,A -85,B 0,C 180,E1 15507.754,E2 15507.754} C_VEL
LIN {X 0,Y 314.065,Z 496.765,A -85,B 0,C 180,E1 15505.657,E2 15505.657} C_VEL
LIN {X 0,Y 311.855,Z 511.758,A -85,B 0,C 180,E1 15503.326,E2 15503.326} C_VEL
LIN {X 0,Y 309.853,Z 525.263,A -85,B 0,C 180,E1 15500.791,E2 15500.791} C_VEL
LIN {X 0,Y 308.07,Z 537.712,A -85,B 0,C 180,E1 15497.959,E2 15497.959} C_VEL
LIN {X 0,Y 306.721,Z 547.954,A -85,B 0,C 180,E1 15495.117,E2 15495.117} C_VEL
LIN {X 0,Y 305.699,Z 556.904,A -85,B 0,C 180,E1 15492.051,E2 15492.051} C_VEL
LIN {X 0,Y 305.042,Z 564.219,A -85,B 0,C 180,E1 15488.862,E2 15488.862} C_VEL
LIN {X 0,Y 304.705,Z 569.73,A -85,B 0,C 180,E1 15485.65,E2 15485.65} C_VEL
LIN {X 0,Y 304.617,Z 573.668,A -85,B 0,C 180,E1 15482.258,E2 15482.258} C_VEL
LIN {X 0,Y 304.726,Z 575.753,A -85,B 0,C 180,E1 15479.06,E2 15479.06} C_VEL
LIN {X 0,Y 305.034,Z 576.272,A -85,B 0,C 180,E1 15475.865,E2 15475.865} C_VEL
LIN {X 0,Y 305.675,Z 575.113,A -85,B 0,C 180,E1 15472.482,E2 15472.482} C_VEL
LIN {X 0,Y 306.772,Z 572.185,A -85,B 0,C 180,E1 15469.104,E2 15469.104} C_VEL
LIN {X 0,Y 308.345,Z 567.777,A -85,B 0,C 180,E1 15465.925,E2 15465.925} C_VEL
LIN {X 0,Y 310.665,Z 561.207,A -85,B 0,C 180,E1 15462.584,E2 15462.584} C_VEL
LIN {X 0,Y 313.727,Z 552.529,A -85,B 0,C 180,E1 15459.283,E2 15459.283} C_VEL
LIN {X 0,Y 317.105,Z 542.804,A -85,B 0,C 180,E1 15456.395,E2 15456.395} C_VEL
LIN {X 0,Y 320.865,Z 531.748,A -85,B 0,C 180,E1 15453.737,E2 15453.737} C_VEL
LIN {X 0,Y 325.199,Z 518.396,A -85,B 0,C 180,E1 15451.138,E2 15451.138} C_VEL
LIN {X 0,Y 329.921,Z 503.165,A -85,B 0,C 180,E1 15448.72,E2 15448.72} C_VEL
LIN {X 0,Y 334.803,Z 486.467,A -85,B 0,C 180,E1 15446.565,E2 15446.565} C_VEL
LIN {X 0,Y 339.732,Z 468.188,A -85,B 0,C 180,E1 15444.668,E2 15444.668} C_VEL
LIN {X 0,Y 344.486,Z 448.948,A -85,B 0,C 180,E1 15443.072,E2 15443.072} C_VEL
LIN {X 0,Y 348.897,Z 428.578,A -85,B 0,C 180,E1 15441.77,E2 15441.77} C_VEL
LIN {X 0,Y 353.173,Z 405.572,A -85,B 0,C 180,E1 15440.682,E2 15440.682} C_VEL
LIN {X 0,Y 367.357,Z 338.881,A -85,B 0,C 180,E1 15438.099,E2 15438.099} C_VEL
LIN {X 0,Y 371.271,Z 322.303,A -85,B 0,C 180,E1 15437.466,E2 15437.466} C_VEL
LIN {X 0,Y 367.929,Z 334,A -85,B 0,C 180,E1 15437.044,E2 15437.044} C_VEL
LIN {X 0,Y 361.205,Z 358.625,A -85,B 0,C 180,E1 15436.146,E2 15436.146} C_VEL
LIN {X 0,Y 355.164,Z 381.822,A -85,B 0,C 180,E1 15435.263,E2 15435.263} C_VEL
LIN {X 0,Y 350.575,Z 400.44,A -85,B 0,C 180,E1 15434.51,E2 15434.51} C_VEL
LIN {X 0,Y 345.758,Z 420.899,A -85,B 0,C 180,E1 15433.721,E2 15433.721} C_VEL
LIN {X 0,Y 343.253,Z 433.502,A -85,B 0,C 180,E1 15433.1,E2 15433.1} C_VEL
LIN {X 0,Y 340.485,Z 453.557,A -85,B 0,C 180,E1 15432.18,E2 15432.18} C_VEL
LIN {X 0,Y 337.072,Z 473.342,A -85,B 0,C 180,E1 15430.963,E2 15430.963} C_VEL
LIN {X 0,Y 333.091,Z 492.958,A -85,B 0,C 180,E1 15429.402,E2 15429.402} C_VEL
LIN {X 0,Y 328.879,Z 511.374,A -85,B 0,C 180,E1 15427.559,E2 15427.559} C_VEL
LIN {X 0,Y 324.634,Z 528.284,A -85,B 0,C 180,E1 15425.485,E2 15425.485} C_VEL
LIN {X 0,Y 320.441,Z 544.298,A -85,B 0,C 180,E1 15423.097,E2 15423.097} C_VEL
LIN {X 0,Y 316.33,Z 559.499,A -85,B 0,C 180,E1 15420.357,E2 15420.357} C_VEL
LIN {X 0,Y 312.51,Z 573.887,A -85,B 0,C 180,E1 15417.197,E2 15417.197} C_VEL
LIN {X 0,Y 309.364,Z 586.461,A -85,B 0,C 180,E1 15413.829,E2 15413.829} C_VEL
LIN {X 0,Y 306.942,Z 597.469,A -85,B 0,C 180,E1 15410.201,E2 15410.201} C_VEL
LIN {X 0,Y 305.377,Z 606.323,A -85,B 0,C 180,E1 15406.551,E2 15406.551} C_VEL
LIN {X 0,Y 304.529,Z 613.257,A -85,B 0,C 180,E1 15402.902,E2 15402.902} C_VEL
LIN {X 0,Y 304.25,Z 618.421,A -85,B 0,C 180,E1 15399.268,E2 15399.268} C_VEL
LIN {X 0,Y 304.28,Z 621.897,A -85,B 0,C 180,E1 15395.659,E2 15395.659} C_VEL
LIN {X 0,Y 304.388,Z 623.663,A -85,B 0,C 180,E1 15392.26,E2 15392.26} C_VEL
LIN {X 0,Y 304.423,Z 623.894,A -85,B 0,C 180,E1 15389.06,E2 15389.06} C_VEL
LIN {X 0,Y 304.322,Z 622.768,A -85,B 0,C 180,E1 15385.667,E2 15385.667} C_VEL
LIN {X 0,Y 304.239,Z 620.091,A -85,B 0,C 180,E1 15382.257,E2 15382.257} C_VEL
LIN {X 0,Y 304.362,Z 615.626,A -85,B 0,C 180,E1 15378.634,E2 15378.634} C_VEL
LIN {X 0,Y 304.988,Z 609.048,A -85,B 0,C 180,E1 15374.797,E2 15374.797} C_VEL
LIN {X 0,Y 306.266,Z 600.895,A -85,B 0,C 180,E1 15371.145,E2 15371.145} C_VEL
LIN {X 0,Y 308.233,Z 591.306,A -85,B 0,C 180,E1 15367.697,E2 15367.697} C_VEL
LIN {X 0,Y 310.834,Z 580.368,A -85,B 0,C 180,E1 15364.468,E2 15364.468} C_VEL
LIN {X 0,Y 314.224,Z 567.253,A -85,B 0,C 180,E1 15361.285,E2 15361.285} C_VEL
LIN {X 0,Y 318.067,Z 552.949,A -85,B 0,C 180,E1 15358.419,E2 15358.419} C_VEL
LIN {X 0,Y 322.228,Z 537.369,A -85,B 0,C 180,E1 15355.833,E2 15355.833} C_VEL
LIN {X 0,Y 326.514,Z 520.738,A -85,B 0,C 180,E1 15353.555,E2 15353.555} C_VEL
LIN {X 0,Y 330.73,Z 503.246,A -85,B 0,C 180,E1 15351.593,E2 15351.593} C_VEL
LIN {X 0,Y 334.936,Z 483.954,A -85,B 0,C 180,E1 15349.85,E2 15349.85} C_VEL
LIN {X 0,Y 338.584,Z 464.66,A -85,B 0,C 180,E1 15348.476,E2 15348.476} C_VEL
LIN {X 0,Y 341.709,Z 444.781,A -85,B 0,C 180,E1 15347.391,E2 15347.391} C_VEL
LIN {X 0,Y 344.201,Z 424.433,A -85,B 0,C 180,E1 15346.589,E2 15346.589} C_VEL
LIN {X 0,Y 345.786,Z 402.698,A -85,B 0,C 180,E1 15346.002,E2 15346.002} C_VEL
LIN {X 0,Y 355.086,Z 216.271,A -85,B 0,C 180,E1 15341.958,E2 15341.958} C_VEL
LIN {X 0,Y 345.333,Z 198.658,A -85,B 0,C 180,E1 15339.755,E2 15339.755} C_VEL
LIN {X 0,Y 335.683,Z 183.14,A -85,B 0,C 180,E1 15337.418,E2 15337.418} C_VEL
LIN {X 0,Y 327.021,Z 170.39,A -85,B 0,C 180,E1 15335.139,E2 15335.139} C_VEL
LIN {X 0,Y 324.11,Z 165.969,A -85,B 0,C 180,E1 15334.235,E2 15334.235} C_VEL
LIN {X 0,Y 318.993,Z 155.333,A -85,B 0,C 180,E1 15330.933,E2 15330.933} C_VEL
LIN {X 0,Y 316.005,Z 149.848,A -85,B 0,C 180,E1 15328.953,E2 15328.953} C_VEL
LIN {X 0,Y 314.027,Z 145.937,A -85,B 0,C 180,E1 15327.495,E2 15327.495} C_VEL
LIN {X 0,Y 312.103,Z 142.28,A -85,B 0,C 180,E1 15326.033,E2 15326.033} C_VEL
LIN {X 0,Y 309.505,Z 137.823,A -85,B 0,C 180,E1 15324.019,E2 15324.019} C_VEL
LIN {X 0,Y 308.963,Z 136.443,A -85,B 0,C 180,E1 15323.456,E2 15323.456} C_VEL
LIN {X 0,Y 306.62,Z 133.113,A -85,B 0,C 180,E1 15321.622,E2 15321.622} C_VEL
LIN {X 0,Y 306.192,Z 131.334,A -85,B 0,C 180,E1 15320.85,E2 15320.85} C_VEL
LIN {X 0,Y 306.215,Z 131.341,A -85,B 0,C 180,E1 15316.271,E2 15316.271} C_VEL
LIN {X 0,Y 306.189,Z 131.315,A -85,B 0,C 180,E1 15311.872,E2 15311.872} C_VEL
LIN {X 0,Y 306.174,Z 131.306,A -85,B 0,C 180,E1 15307.505,E2 15307.505} C_VEL
LIN {X 0,Y 306.185,Z 131.329,A -85,B 0,C 180,E1 15302.995,E2 15302.995} C_VEL
LIN {X 0,Y 306.207,Z 131.333,A -85,B 0,C 180,E1 15298.503,E2 15298.503} C_VEL
LIN {X 0,Y 306.185,Z 131.305,A -85,B 0,C 180,E1 15294.001,E2 15294.001} C_VEL
LIN {X 0,Y 306.172,Z 131.314,A -85,B 0,C 180,E1 15289.462,E2 15289.462} C_VEL
LIN {X 0,Y 306.184,Z 131.345,A -85,B 0,C 180,E1 15285.049,E2 15285.049} C_VEL
LIN {X 0,Y 306.201,Z 131.324,A -85,B 0,C 180,E1 15280.545,E2 15280.545} C_VEL
LIN {X 0,Y 306.18,Z 131.311,A -85,B 0,C 180,E1 15276.112,E2 15276.112} C_VEL
LIN {X 0,Y 306.229,Z 131.54,A -85,B 0,C 180,E1 15274.573,E2 15274.573} C_VEL
LIN {X 0,Y 307.624,Z 134.99,A -85,B 0,C 180,E1 15272.942,E2 15272.942} C_VEL
LIN {X 0,Y 309.067,Z 136.956,A -85,B 0,C 180,E1 15271.814,E2 15271.814} C_VEL
LIN {X 0,Y 311.239,Z 141.065,A -85,B 0,C 180,E1 15269.923,E2 15269.923} C_VEL
LIN {X 0,Y 314.221,Z 146.942,A -85,B 0,C 180,E1 15267.468,E2 15267.468} C_VEL
LIN {X 0,Y 318.242,Z 154.955,A -85,B 0,C 180,E1 15264.459,E2 15264.459} C_VEL
LIN {X 0,Y 323.551,Z 166.698,A -85,B 0,C 180,E1 15260.69,E2 15260.69} C_VEL
LIN {X 0,Y 325.837,Z 171.941,A -85,B 0,C 180,E1 15259.243,E2 15259.243} C_VEL
LIN {X 0,Y 334.795,Z 185.592,A -85,B 0,C 180,E1 15256.879,E2 15256.879} C_VEL
LIN {X 0,Y 344.134,Z 201.198,A -85,B 0,C 180,E1 15254.615,E2 15254.615} C_VEL
LIN {X 0,Y 352.343,Z 216.468,A -85,B 0,C 180,E1 15252.762,E2 15252.762} C_VEL
LIN {X 0,Y 353.216,Z 225.131,A -85,B 0,C 180,E1 15252.384,E2 15252.384} C_VEL
LIN {X 0,Y 346.169,Z 396.124,A -85,B 0,C 180,E1 15248.997,E2 15248.997} C_VEL
LIN {X 0,Y 344.473,Z 415.551,A -85,B 0,C 180,E1 15248.332,E2 15248.332} C_VEL
LIN {X 0,Y 342.161,Z 433.689,A -85,B 0,C 180,E1 15247.43,E2 15247.43} C_VEL
LIN {X 0,Y 339.082,Z 452.022,A -85,B 0,C 180,E1 15246.204,E2 15246.204} C_VEL
LIN {X 0,Y 335.464,Z 469.459,A -85,B 0,C 180,E1 15244.698,E2 15244.698} C_VEL
LIN {X 0,Y 331.437,Z 486.063,A -85,B 0,C 180,E1 15242.887,E2 15242.887} C_VEL
LIN {X 0,Y 327.174,Z 501.524,A -85,B 0,C 180,E1 15240.788,E2 15240.788} C_VEL
LIN {X 0,Y 322.956,Z 515.504,A -85,B 0,C 180,E1 15238.447,E2 15238.447} C_VEL
LIN {X 0,Y 318.879,Z 528.18,A -85,B 0,C 180,E1 15235.837,E2 15235.837} C_VEL
LIN {X 0,Y 315.11,Z 539.469,A -85,B 0,C 180,E1 15232.971,E2 15232.971} C_VEL
LIN {X 0,Y 311.815,Z 549.288,A -85,B 0,C 180,E1 15229.869,E2 15229.869} C_VEL
LIN {X 0,Y 309.109,Z 557.621,A -85,B 0,C 180,E1 15226.537,E2 15226.537} C_VEL
LIN {X 0,Y 307.05,Z 564.428,A -85,B 0,C 180,E1 15222.983,E2 15222.983} C_VEL
LIN {X 0,Y 305.678,Z 569.61,A -85,B 0,C 180,E1 15219.222,E2 15219.222} C_VEL
LIN {X 0,Y 304.939,Z 572.938,A -85,B 0,C 180,E1 15215.455,E2 15215.455} C_VEL
LIN {X 0,Y 304.653,Z 574.544,A -85,B 0,C 180,E1 15211.691,E2 15211.691} C_VEL
LIN {X 0,Y 304.658,Z 574.536,A -85,B 0,C 180,E1 15208.118,E2 15208.118} C_VEL
LIN {X 0,Y 304.953,Z 572.895,A -85,B 0,C 180,E1 15204.354,E2 15204.354} C_VEL
LIN {X 0,Y 305.709,Z 569.523,A -85,B 0,C 180,E1 15200.587,E2 15200.587} C_VEL
LIN {X 0,Y 307.101,Z 564.284,A -85,B 0,C 180,E1 15196.825,E2 15196.825} C_VEL
LIN {X 0,Y 309.186,Z 557.432,A -85,B 0,C 180,E1 15193.272,E2 15193.272} C_VEL
LIN {X 0,Y 311.953,Z 548.945,A -85,B 0,C 180,E1 15189.904,E2 15189.904} C_VEL
LIN {X 0,Y 315.238,Z 539.176,A -85,B 0,C 180,E1 15186.839,E2 15186.839} C_VEL
LIN {X 0,Y 319.034,Z 527.825,A -85,B 0,C 180,E1 15183.974,E2 15183.974} C_VEL
LIN {X 0,Y 323.174,Z 514.954,A -85,B 0,C 180,E1 15181.343,E2 15181.343} C_VEL
LIN {X 0,Y 327.541,Z 500.433,A -85,B 0,C 180,E1 15178.942,E2 15178.942} C_VEL
LIN {X 0,Y 331.662,Z 485.437,A -85,B 0,C 180,E1 15176.929,E2 15176.929} C_VEL
LIN {X 0,Y 331.986,Z 484.102,A -85,B 0,C 180,E1 15176.774,E2 15176.774} C_VEL
LIN {X 0,Y 332.766,Z 477.989,A -85,B 0,C 180,E1 15175.97,E2 15175.97} C_VEL
LIN {X 0,Y 331.656,Z 462.368,A -85,B 0,C 180,E1 15173.779,E2 15173.779} C_VEL
LIN {X 0,Y 332.22,Z 455.729,A -85,B 0,C 180,E1 15173.102,E2 15173.102} C_VEL
LIN {X 0,Y 335.337,Z 438.764,A -85,B 0,C 180,E1 15171.887,E2 15171.887} C_VEL
LIN {X 0,Y 338.061,Z 419.583,A -85,B 0,C 180,E1 15170.848,E2 15170.848} C_VEL
LIN {X 0,Y 339.988,Z 400.136,A -85,B 0,C 180,E1 15170.118,E2 15170.118} C_VEL
LIN {X 0,Y 341.315,Z 374.478,A -85,B 0,C 180,E1 15169.532,E2 15169.532} C_VEL
LIN {X 0,Y 347.613,Z 224.531,A -85,B 0,C 180,E1 15166.539,E2 15166.539} C_VEL
LIN {X 0,Y 346.891,Z 219.835,A -85,B 0,C 180,E1 15166.282,E2 15166.282} C_VEL
LIN {X 0,Y 337.893,Z 203.272,A -85,B 0,C 180,E1 15164.147,E2 15164.147} C_VEL
LIN {X 0,Y 331.009,Z 191.819,A -85,B 0,C 180,E1 15162.405,E2 15162.405} C_VEL
LIN {X 0,Y 328.236,Z 192.698,A -85,B 0,C 180,E1 15161.845,E2 15161.845} C_VEL
LIN {X 0,Y 325.546,Z 194.746,A -85,B 0,C 180,E1 15161.326,E2 15161.326} C_VEL
LIN {X 0,Y 323.448,Z 194.816,A -85,B 0,C 180,E1 15160.835,E2 15160.835} C_VEL
LIN {X 0,Y 326.291,Z 201.69,A -85,B 0,C 180,E1 15160.268,E2 15160.268} C_VEL
LIN {X 0,Y 327.844,Z 219.863,A -85,B 0,C 180,E1 15159.443,E2 15159.443} C_VEL
LIN {X 0,Y 316.601,Z 404.327,A -85,B 0,C 180,E1 15153.884,E2 15153.884} C_VEL
LIN {X 0,Y 315.099,Z 424.574,A -85,B 0,C 180,E1 15152.916,E2 15152.916} C_VEL
LIN {X 0,Y 313.259,Z 443.683,A -85,B 0,C 180,E1 15151.672,E2 15151.672} C_VEL
LIN {X 0,Y 310.998,Z 463.265,A -85,B 0,C 180,E1 15150.022,E2 15150.022} C_VEL
LIN {X 0,Y 308.755,Z 480.366,A -85,B 0,C 180,E1 15148.217,E2 15148.217} C_VEL
LIN {X 0,Y 306.343,Z 497.169,A -85,B 0,C 180,E1 15146.035,E2 15146.035} C_VEL
LIN {X 0,Y 304.062,Z 512.201,A -85,B 0,C 180,E1 15143.652,E2 15143.652} C_VEL
LIN {X 0,Y 301.916,Z 526.289,A -85,B 0,C 180,E1 15140.946,E2 15140.946} C_VEL
LIN {X 0,Y 300.1,Z 538.677,A -85,B 0,C 180,E1 15138.051,E2 15138.051} C_VEL
LIN {X 0,Y 298.723,Z 548.901,A -85,B 0,C 180,E1 15135.134,E2 15135.134} C_VEL
LIN {X 0,Y 297.695,Z 557.722,A -85,B 0,C 180,E1 15132.019,E2 15132.019} C_VEL
LIN {X 0,Y 297.029,Z 565.082,A -85,B 0,C 180,E1 15128.713,E2 15128.713} C_VEL
LIN {X 0,Y 296.703,Z 570.561,A -85,B 0,C 180,E1 15125.415,E2 15125.415} C_VEL
LIN {X 0,Y 296.634,Z 574.33,A -85,B 0,C 180,E1 15122.125,E2 15122.125} C_VEL
LIN {X 0,Y 296.763,Z 576.488,A -85,B 0,C 180,E1 15118.842,E2 15118.842} C_VEL
LIN {X 0,Y 297.141,Z 577.052,A -85,B 0,C 180,E1 15115.368,E2 15115.368} C_VEL
LIN {X 0,Y 297.892,Z 575.871,A -85,B 0,C 180,E1 15111.896,E2 15111.896} C_VEL
LIN {X 0,Y 299.15,Z 572.957,A -85,B 0,C 180,E1 15108.432,E2 15108.432} C_VEL
LIN {X 0,Y 301.047,Z 568.227,A -85,B 0,C 180,E1 15104.986,E2 15104.986} C_VEL
LIN {X 0,Y 303.674,Z 561.567,A -85,B 0,C 180,E1 15101.574,E2 15101.574} C_VEL
LIN {X 0,Y 306.675,Z 553.903,A -85,B 0,C 180,E1 15098.583,E2 15098.583} C_VEL
LIN {X 0,Y 310.588,Z 543.747,A -85,B 0,C 180,E1 15095.463,E2 15095.463} C_VEL
LIN {X 0,Y 314.965,Z 531.995,A -85,B 0,C 180,E1 15092.594,E2 15092.594} C_VEL
LIN {X 0,Y 319.706,Z 518.719,A -85,B 0,C 180,E1 15089.975,E2 15089.975} C_VEL
LIN {X 0,Y 325.131,Z 502.937,A -85,B 0,C 180,E1 15087.441,E2 15087.441} C_VEL
LIN {X 0,Y 330.384,Z 486.61,A -85,B 0,C 180,E1 15085.323,E2 15085.323} C_VEL
LIN {X 0,Y 335.998,Z 467.936,A -85,B 0,C 180,E1 15083.37,E2 15083.37} C_VEL
LIN {X 0,Y 341.183,Z 449.077,A -85,B 0,C 180,E1 15081.805,E2 15081.805} C_VEL
LIN {X 0,Y 346.013,Z 429.174,A -85,B 0,C 180,E1 15080.527,E2 15080.527} C_VEL
LIN {X 0,Y 350.984,Z 405.393,A -85,B 0,C 180,E1 15079.402,E2 15079.402} C_VEL
LIN {X 0,Y 362.136,Z 356.735,A -85,B 0,C 180,E1 15077.494,E2 15077.494} C_VEL
LIN {X 0,Y 356.442,Z 376.767,A -85,B 0,C 180,E1 15076.758,E2 15076.758} C_VEL
LIN {X 0,Y 350.03,Z 400.365,A -85,B 0,C 180,E1 15075.866,E2 15075.866} C_VEL
LIN {X 0,Y 343.907,Z 424.171,A -85,B 0,C 180,E1 15074.921,E2 15074.921} C_VEL
LIN {X 0,Y 337.093,Z 449.162,A -85,B 0,C 180,E1 15073.601,E2 15073.601} C_VEL
LIN {X 0,Y 332.347,Z 465.468,A -85,B 0,C 180,E1 15072.37,E2 15072.37} C_VEL
LIN {X 0,Y 327.896,Z 487.228,A -85,B 0,C 180,E1 15070.736,E2 15070.736} C_VEL
LIN {X 0,Y 323.568,Z 505.811,A -85,B 0,C 180,E1 15068.965,E2 15068.965} C_VEL
LIN {X 0,Y 319.222,Z 522.767,A -85,B 0,C 180,E1 15066.97,E2 15066.97} C_VEL
LIN {X 0,Y 314.798,Z 538.974,A -85,B 0,C 180,E1 15064.65,E2 15064.65} C_VEL
LIN {X 0,Y 310.329,Z 554.787,A -85,B 0,C 180,E1 15061.898,E2 15061.898} C_VEL
LIN {X 0,Y 306.291,Z 569.007,A -85,B 0,C 180,E1 15058.891,E2 15058.891} C_VEL
LIN {X 0,Y 302.83,Z 581.723,A -85,B 0,C 180,E1 15055.629,E2 15055.629} C_VEL
LIN {X 0,Y 300.065,Z 592.909,A -85,B 0,C 180,E1 15052.131,E2 15052.131} C_VEL
LIN {X 0,Y 298.12,Z 602.158,A -85,B 0,C 180,E1 15048.581,E2 15048.581} C_VEL
LIN {X 0,Y 296.888,Z 609.916,A -85,B 0,C 180,E1 15044.831,E2 15044.831} C_VEL
LIN {X 0,Y 296.338,Z 615.807,A -85,B 0,C 180,E1 15041.089,E2 15041.089} C_VEL
LIN {X 0,Y 296.253,Z 619.976,A -85,B 0,C 180,E1 15037.37,E2 15037.37} C_VEL
LIN {X 0,Y 296.361,Z 622.412,A -85,B 0,C 180,E1 15033.87,E2 15033.87} C_VEL
LIN {X 0,Y 296.449,Z 623.299,A -85,B 0,C 180,E1 15030.581,E2 15030.581} C_VEL
LIN {X 0,Y 296.398,Z 622.787,A -85,B 0,C 180,E1 15027.101,E2 15027.101} C_VEL
LIN {X 0,Y 296.27,Z 620.841,A -85,B 0,C 180,E1 15023.607,E2 15023.607} C_VEL
LIN {X 0,Y 296.275,Z 617.296,A -85,B 0,C 180,E1 15020.091,E2 15020.091} C_VEL
LIN {X 0,Y 296.647,Z 611.914,A -85,B 0,C 180,E1 15016.354,E2 15016.354} C_VEL
LIN {X 0,Y 297.673,Z 604.603,A -85,B 0,C 180,E1 15012.54,E2 15012.54} C_VEL
LIN {X 0,Y 299.435,Z 595.644,A -85,B 0,C 180,E1 15008.863,E2 15008.863} C_VEL
LIN {X 0,Y 301.969,Z 585.037,A -85,B 0,C 180,E1 15005.343,E2 15005.343} C_VEL
LIN {X 0,Y 305.189,Z 572.992,A -85,B 0,C 180,E1 15002.065,E2 15002.065} C_VEL
LIN {X 0,Y 309.234,Z 558.572,A -85,B 0,C 180,E1 14998.848,E2 14998.848} C_VEL
LIN {X 0,Y 313.754,Z 542.668,A -85,B 0,C 180,E1 14995.95,E2 14995.95} C_VEL
LIN {X 0,Y 318.317,Z 526.067,A -85,B 0,C 180,E1 14993.472,E2 14993.472} C_VEL
LIN {X 0,Y 323.056,Z 507.761,A -85,B 0,C 180,E1 14991.255,E2 14991.255} C_VEL
LIN {X 0,Y 327.446,Z 488.997,A -85,B 0,C 180,E1 14989.43,E2 14989.43} C_VEL
LIN {X 0,Y 331.395,Z 469.758,A -85,B 0,C 180,E1 14987.95,E2 14987.95} C_VEL
LIN {X 0,Y 334.646,Z 450.962,A -85,B 0,C 180,E1 14986.829,E2 14986.829} C_VEL
LIN {X 0,Y 337.46,Z 430.503,A -85,B 0,C 180,E1 14985.92,E2 14985.92} C_VEL
LIN {X 0,Y 339.417,Z 409.212,A -85,B 0,C 180,E1 14985.268,E2 14985.268} C_VEL
LIN {X 0,Y 349.327,Z 219.485,A -85,B 0,C 180,E1 14981.098,E2 14981.098} C_VEL
LIN {X 0,Y 340.126,Z 202.845,A -85,B 0,C 180,E1 14978.928,E2 14978.928} C_VEL
LIN {X 0,Y 331.424,Z 188.676,A -85,B 0,C 180,E1 14976.733,E2 14976.733} C_VEL
LIN {X 0,Y 323.053,Z 176.176,A -85,B 0,C 180,E1 14974.445,E2 14974.445} C_VEL
LIN {X 0,Y 316.146,Z 166.236,A -85,B 0,C 180,E1 14972.309,E2 14972.309} C_VEL
LIN {X 0,Y 311.369,Z 156.567,A -85,B 0,C 180,E1 14969.005,E2 14969.005} C_VEL
LIN {X 0,Y 308.602,Z 151.494,A -85,B 0,C 180,E1 14967.005,E2 14967.005} C_VEL
LIN {X 0,Y 306.5,Z 147.361,A -85,B 0,C 180,E1 14965.299,E2 14965.299} C_VEL
LIN {X 0,Y 304.484,Z 143.666,A -85,B 0,C 180,E1 14963.617,E2 14963.617} C_VEL
LIN {X 0,Y 303.57,Z 142.207,A -85,B 0,C 180,E1 14962.87,E2 14962.87} C_VEL
LIN {X 0,Y 301.537,Z 138.516,A -85,B 0,C 180,E1 14960.984,E2 14960.984} C_VEL
LIN {X 0,Y 301.01,Z 137.401,A -85,B 0,C 180,E1 14960.412,E2 14960.412} C_VEL
LIN {X 0,Y 298.781,Z 134.285,A -85,B 0,C 180,E1 14958.334,E2 14958.334} C_VEL
LIN {X 0,Y 298.242,Z 132.309,A -85,B 0,C 180,E1 14957.36,E2 14957.36} C_VEL
LIN {X 0,Y 298.252,Z 132.294,A -85,B 0,C 180,E1 14952.783,E2 14952.783} C_VEL
LIN {X 0,Y 298.27,Z 132.297,A -85,B 0,C 180,E1 14948.287,E2 14948.287} C_VEL
LIN {X 0,Y 298.247,Z 132.335,A -85,B 0,C 180,E1 14943.844,E2 14943.844} C_VEL
LIN {X 0,Y 298.237,Z 132.308,A -85,B 0,C 180,E1 14939.231,E2 14939.231} C_VEL
LIN {X 0,Y 298.258,Z 132.29,A -85,B 0,C 180,E1 14934.614,E2 14934.614} C_VEL
LIN {X 0,Y 298.251,Z 132.31,A -85,B 0,C 180,E1 14930.155,E2 14930.155} C_VEL
LIN {X 0,Y 298.236,Z 132.334,A -85,B 0,C 180,E1 14925.635,E2 14925.635} C_VEL
LIN {X 0,Y 298.248,Z 132.305,A -85,B 0,C 180,E1 14920.972,E2 14920.972} C_VEL
LIN {X 0,Y 298.247,Z 132.327,A -85,B 0,C 180,E1 14918.153,E2 14918.153} C_VEL
LIN {X 0,Y 299.618,Z 135.883,A -85,B 0,C 180,E1 14916.184,E2 14916.184} C_VEL
LIN {X 0,Y 301.216,Z 137.668,A -85,B 0,C 180,E1 14914.856,E2 14914.856} C_VEL
LIN {X 0,Y 302.734,Z 141.27,A -85,B 0,C 180,E1 14913.09,E2 14913.09} C_VEL
LIN {X 0,Y 303.928,Z 142.828,A -85,B 0,C 180,E1 14912.15,E2 14912.15} C_VEL
LIN {X 0,Y 305.995,Z 146.982,A -85,B 0,C 180,E1 14910.22,E2 14910.22} C_VEL
LIN {X 0,Y 309.067,Z 153.17,A -85,B 0,C 180,E1 14907.6,E2 14907.6} C_VEL
LIN {X 0,Y 312.885,Z 160.872,A -85,B 0,C 180,E1 14904.661,E2 14904.661} C_VEL
LIN {X 0,Y 317.754,Z 171.635,A -85,B 0,C 180,E1 14901.173,E2 14901.173} C_VEL
LIN {X 0,Y 327.565,Z 186.373,A -85,B 0,C 180,E1 14898.373,E2 14898.373} C_VEL
LIN {X 0,Y 336.699,Z 201.32,A -85,B 0,C 180,E1 14896.011,E2 14896.011} C_VEL
LIN {X 0,Y 345.83,Z 217.963,A -85,B 0,C 180,E1 14893.833,E2 14893.833} C_VEL
LIN {X 0,Y 347.085,Z 220.854,A -85,B 0,C 180,E1 14893.533,E2 14893.533} C_VEL
LIN {X 0,Y 347.548,Z 226.725,A -85,B 0,C 180,E1 14893.289,E2 14893.289} C_VEL
LIN {X 0,Y 340.204,Z 396.423,A -85,B 0,C 180,E1 14889.886,E2 14889.886} C_VEL
LIN {X 0,Y 338.438,Z 415.883,A -85,B 0,C 180,E1 14889.213,E2 14889.213} C_VEL
LIN {X 0,Y 335.902,Z 434.846,A -85,B 0,C 180,E1 14888.252,E2 14888.252} C_VEL
LIN {X 0,Y 332.785,Z 452.638,A -85,B 0,C 180,E1 14887.041,E2 14887.041} C_VEL
LIN {X 0,Y 328.956,Z 470.333,A -85,B 0,C 180,E1 14885.487,E2 14885.487} C_VEL
LIN {X 0,Y 324.772,Z 486.863,A -85,B 0,C 180,E1 14883.651,E2 14883.651} C_VEL
LIN {X 0,Y 320.342,Z 502.276,A -85,B 0,C 180,E1 14881.519,E2 14881.519} C_VEL
LIN {X 0,Y 315.944,Z 516.23,A -85,B 0,C 180,E1 14879.137,E2 14879.137} C_VEL
LIN {X 0,Y 311.687,Z 528.88,A -85,B 0,C 180,E1 14876.479,E2 14876.479} C_VEL
LIN {X 0,Y 307.742,Z 540.154,A -85,B 0,C 180,E1 14873.554,E2 14873.554} C_VEL
LIN {X 0,Y 304.096,Z 550.467,A -85,B 0,C 180,E1 14870.195,E2 14870.195} C_VEL
LIN {X 0,Y 301.285,Z 558.686,A -85,B 0,C 180,E1 14866.78,E2 14866.78} C_VEL
LIN {X 0,Y 299.145,Z 565.378,A -85,B 0,C 180,E1 14863.136,E2 14863.136} C_VEL
LIN {X 0,Y 297.777,Z 570.26,A -85,B 0,C 180,E1 14859.469,E2 14859.469} C_VEL
LIN {X 0,Y 296.987,Z 573.585,A -85,B 0,C 180,E1 14855.602,E2 14855.602} C_VEL
LIN {X 0,Y 296.681,Z 575.189,A -85,B 0,C 180,E1 14851.737,E2 14851.737} C_VEL
LIN {X 0,Y 296.686,Z 575.181,A -85,B 0,C 180,E1 14848.067,E2 14848.067} C_VEL
LIN {X 0,Y 297.002,Z 573.542,A -85,B 0,C 180,E1 14844.202,E2 14844.202} C_VEL
LIN {X 0,Y 297.812,Z 570.172,A -85,B 0,C 180,E1 14840.335,E2 14840.335} C_VEL
LIN {X 0,Y 299.296,Z 564.94,A -85,B 0,C 180,E1 14836.475,E2 14836.475} C_VEL
LIN {X 0,Y 301.504,Z 558.094,A -85,B 0,C 180,E1 14832.833,E2 14832.833} C_VEL
LIN {X 0,Y 304.394,Z 549.708,A -85,B 0,C 180,E1 14829.417,E2 14829.417} C_VEL
LIN {X 0,Y 307.879,Z 539.86,A -85,B 0,C 180,E1 14826.252,E2 14826.252} C_VEL
LIN {X 0,Y 311.854,Z 528.527,A -85,B 0,C 180,E1 14823.328,E2 14823.328} C_VEL
LIN {X 0,Y 316.331,Z 515.192,A -85,B 0,C 180,E1 14820.559,E2 14820.559} C_VEL
LIN {X 0,Y 320.73,Z 501.199,A -85,B 0,C 180,E1 14818.206,E2 14818.206} C_VEL
LIN {X 0,Y 325.195,Z 485.539,A -85,B 0,C 180,E1 14816.078,E2 14816.078} C_VEL
LIN {X 0,Y 329.216,Z 469.571,A -85,B 0,C 180,E1 14814.329,E2 14814.329} C_VEL
LIN {X 0,Y 332.22,Z 455.729,A -85,B 0,C 180,E1 14813.102,E2 14813.102} C_VEL
LIN {X 0,Y 332.828,Z 448.938,A -85,B 0,C 180,E1 14812.459,E2 14812.459} C_VEL
LIN {X 0,Y 331.299,Z 432.82,A -85,B 0,C 180,E1 14810.741,E2 14810.741} C_VEL
LIN {X 0,Y 331.394,Z 425.696,A -85,B 0,C 180,E1 14810.214,E2 14810.214} C_VEL
LIN {X 0,Y 331.515,Z 424.642,A -85,B 0,C 180,E1 14810.159,E2 14810.159} C_VEL
LIN {X 0,Y 333.715,Z 405.248,A -85,B 0,C 180,E1 14809.346,E2 14809.346} C_VEL
LIN {X 0,Y 335.063,Z 384.945,A -85,B 0,C 180,E1 14808.809,E2 14808.809} C_VEL
LIN {X 0,Y 342.058,Z 225.865,A -85,B 0,C 180,E1 14805.596,E2 14805.596} C_VEL
LIN {X 0,Y 341.546,Z 223.565,A -85,B 0,C 180,E1 14805.437,E2 14805.437} C_VEL
LIN {X 0,Y 332.938,Z 207.566,A -85,B 0,C 180,E1 14803.302,E2 14803.302} C_VEL
LIN {X 0,Y 328.954,Z 200.713,A -85,B 0,C 180,E1 14802.26,E2 14802.26} C_VEL
LIN {X 0,Y 326.089,Z 202.72,A -85,B 0,C 180,E1 14801.711,E2 14801.711} C_VEL
LIN {X 0,Y 322.884,Z 208.879,A -85,B 0,C 180,E1 14801.21,E2 14801.21} C_VEL
LIN {X 0,Y 321.039,Z 210.459,A -85,B 0,C 180,E1 14800.847,E2 14800.847} C_VEL
LIN {X 0,Y 320.125,Z 210.466,A -85,B 0,C 180,E1 14800.616,E2 14800.616} C_VEL
LIN {X 0,Y 320.896,Z 220.949,A -85,B 0,C 180,E1 14800.135,E2 14800.135} C_VEL
LIN {X 0,Y 309.196,Z 405.039,A -85,B 0,C 180,E1 14794.431,E2 14794.431} C_VEL
LIN {X 0,Y 307.626,Z 425.371,A -85,B 0,C 180,E1 14793.43,E2 14793.43} C_VEL
LIN {X 0,Y 305.694,Z 444.691,A -85,B 0,C 180,E1 14792.137,E2 14792.137} C_VEL
LIN {X 0,Y 303.425,Z 463.706,A -85,B 0,C 180,E1 14790.496,E2 14790.496} C_VEL
LIN {X 0,Y 301.02,Z 481.451,A -85,B 0,C 180,E1 14788.575,E2 14788.575} C_VEL
LIN {X 0,Y 298.537,Z 498.109,A -85,B 0,C 180,E1 14786.345,E2 14786.345} C_VEL
LIN {X 0,Y 296.189,Z 513.123,A -85,B 0,C 180,E1 14783.897,E2 14783.897} C_VEL
LIN {X 0,Y 293.992,Z 527.117,A -85,B 0,C 180,E1 14781.132,E2 14781.132} C_VEL
LIN {X 0,Y 292.125,Z 539.529,A -85,B 0,C 180,E1 14778.148,E2 14778.148} C_VEL
LIN {X 0,Y 290.641,Z 550.374,A -85,B 0,C 180,E1 14774.953,E2 14774.953} C_VEL
LIN {X 0,Y 289.627,Z 559.063,A -85,B 0,C 180,E1 14771.753,E2 14771.753} C_VEL
LIN {X 0,Y 288.987,Z 566.267,A -85,B 0,C 180,E1 14768.356,E2 14768.356} C_VEL
LIN {X 0,Y 288.692,Z 571.637,A -85,B 0,C 180,E1 14764.968,E2 14764.968} C_VEL
LIN {X 0,Y 288.655,Z 575.287,A -85,B 0,C 180,E1 14761.588,E2 14761.588} C_VEL
LIN {X 0,Y 288.831,Z 577.342,A -85,B 0,C 180,E1 14758.215,E2 14758.215} C_VEL
LIN {X 0,Y 289.266,Z 577.841,A -85,B 0,C 180,E1 14754.844,E2 14754.844} C_VEL
LIN {X 0,Y 290.141,Z 576.67,A -85,B 0,C 180,E1 14751.279,E2 14751.279} C_VEL
LIN {X 0,Y 291.575,Z 573.764,A -85,B 0,C 180,E1 14747.725,E2 14747.725} C_VEL
LIN {X 0,Y 293.705,Z 569.046,A -85,B 0,C 180,E1 14744.197,E2 14744.197} C_VEL
LIN {X 0,Y 296.625,Z 562.465,A -85,B 0,C 180,E1 14740.711,E2 14740.711} C_VEL
LIN {X 0,Y 300.39,Z 553.817,A -85,B 0,C 180,E1 14737.288,E2 14737.288} C_VEL
LIN {X 0,Y 304.752,Z 543.501,A -85,B 0,C 180,E1 14734.129,E2 14734.129} C_VEL
LIN {X 0,Y 309.595,Z 531.659,A -85,B 0,C 180,E1 14731.236,E2 14731.236} C_VEL
LIN {X 0,Y 315.211,Z 517.488,A -85,B 0,C 180,E1 14728.441,E2 14728.441} C_VEL
LIN {X 0,Y 320.978,Z 502.162,A -85,B 0,C 180,E1 14726.003,E2 14726.003} C_VEL
LIN {X 0,Y 327.202,Z 484.679,A -85,B 0,C 180,E1 14723.762,E2 14723.762} C_VEL
LIN {X 0,Y 333.158,Z 466.795,A -85,B 0,C 180,E1 14721.922,E2 14721.922} C_VEL
LIN {X 0,Y 339.113,Z 447.202,A -85,B 0,C 180,E1 14720.332,E2 14720.332} C_VEL
LIN {X 0,Y 344.087,Z 428.67,A -85,B 0,C 180,E1 14719.171,E2 14719.171} C_VEL
LIN {X 0,Y 350.317,Z 401.846,A -85,B 0,C 180,E1 14717.946,E2 14717.946} C_VEL
LIN {X 0,Y 352.627,Z 392.272,A -85,B 0,C 180,E1 14717.55,E2 14717.55} C_VEL
LIN {X 0,Y 347.877,Z 408.73,A -85,B 0,C 180,E1 14716.906,E2 14716.906} C_VEL
LIN {X 0,Y 342.52,Z 427.781,A -85,B 0,C 180,E1 14716.125,E2 14716.125} C_VEL
LIN {X 0,Y 335.142,Z 451.22,A -85,B 0,C 180,E1 14714.877,E2 14714.877} C_VEL
LIN {X 0,Y 329.625,Z 467.376,A -85,B 0,C 180,E1 14713.638,E2 14713.638} C_VEL
LIN {X 0,Y 323.548,Z 484.408,A -85,B 0,C 180,E1 14712.114,E2 14712.114} C_VEL
LIN {X 0,Y 318.495,Z 499.982,A -85,B 0,C 180,E1 14710.413,E2 14710.413} C_VEL
LIN {X 0,Y 313.781,Z 518.006,A -85,B 0,C 180,E1 14708.384,E2 14708.384} C_VEL
LIN {X 0,Y 309.071,Z 534.738,A -85,B 0,C 180,E1 14706.072,E2 14706.072} C_VEL
LIN {X 0,Y 304.377,Z 550.651,A -85,B 0,C 180,E1 14703.384,E2 14703.384} C_VEL
LIN {X 0,Y 299.811,Z 565.854,A -85,B 0,C 180,E1 14700.238,E2 14700.238} C_VEL
LIN {X 0,Y 295.949,Z 579.097,A -85,B 0,C 180,E1 14696.885,E2 14696.885} C_VEL
LIN {X 0,Y 292.701,Z 591.143,A -85,B 0,C 180,E1 14693.132,E2 14693.132} C_VEL
LIN {X 0,Y 290.417,Z 601.019,A -85,B 0,C 180,E1 14689.301,E2 14689.301} C_VEL
LIN {X 0,Y 289.031,Z 608.86,A -85,B 0,C 180,E1 14685.45,E2 14685.45} C_VEL
LIN {X 0,Y 288.384,Z 614.866,A -85,B 0,C 180,E1 14681.602,E2 14681.602} C_VEL
LIN {X 0,Y 288.263,Z 619.146,A -85,B 0,C 180,E1 14677.776,E2 14677.776} C_VEL
LIN {X 0,Y 288.368,Z 621.687,A -85,B 0,C 180,E1 14674.177,E2 14674.177} C_VEL
LIN {X 0,Y 288.475,Z 622.63,A -85,B 0,C 180,E1 14670.796,E2 14670.796} C_VEL
LIN {X 0,Y 288.424,Z 622.216,A -85,B 0,C 180,E1 14667.219,E2 14667.219} C_VEL
LIN {X 0,Y 288.291,Z 620.46,A -85,B 0,C 180,E1 14663.829,E2 14663.829} C_VEL
LIN {X 0,Y 288.279,Z 617.089,A -85,B 0,C 180,E1 14660.216,E2 14660.216} C_VEL
LIN {X 0,Y 288.639,Z 611.902,A -85,B 0,C 180,E1 14656.377,E2 14656.377} C_VEL
LIN {X 0,Y 289.658,Z 604.936,A -85,B 0,C 180,E1 14652.525,E2 14652.525} C_VEL
LIN {X 0,Y 291.498,Z 596.044,A -85,B 0,C 180,E1 14648.681,E2 14648.681} C_VEL
LIN {X 0,Y 294.117,Z 585.633,A -85,B 0,C 180,E1 14645.07,E2 14645.07} C_VEL
LIN {X 0,Y 297.444,Z 573.763,A -85,B 0,C 180,E1 14641.709,E2 14641.709} C_VEL
LIN {X 0,Y 301.354,Z 560.501,A -85,B 0,C 180,E1 14638.608,E2 14638.608} C_VEL
LIN {X 0,Y 305.753,Z 545.83,A -85,B 0,C 180,E1 14635.775,E2 14635.775} C_VEL
LIN {X 0,Y 310.45,Z 529.654,A -85,B 0,C 180,E1 14633.2,E2 14633.2} C_VEL
LIN {X 0,Y 315.395,Z 511.764,A -85,B 0,C 180,E1 14630.888,E2 14630.888} C_VEL
LIN {X 0,Y 319.955,Z 493.553,A -85,B 0,C 180,E1 14628.987,E2 14628.987} C_VEL
LIN {X 0,Y 324.21,Z 474.394,A -85,B 0,C 180,E1 14627.397,E2 14627.397} C_VEL
LIN {X 0,Y 327.784,Z 455.609,A -85,B 0,C 180,E1 14626.179,E2 14626.179} C_VEL
LIN {X 0,Y 330.86,Z 435.625,A -85,B 0,C 180,E1 14625.205,E2 14625.205} C_VEL
LIN {X 0,Y 333.181,Z 414.191,A -85,B 0,C 180,E1 14624.472,E2 14624.472} C_VEL
LIN {X 0,Y 343.647,Z 222.69,A -85,B 0,C 180,E1 14620.207,E2 14620.207} C_VEL
LIN {X 0,Y 333.956,Z 205.112,A -85,B 0,C 180,E1 14617.808,E2 14617.808} C_VEL
LIN {X 0,Y 323.957,Z 189.037,A -85,B 0,C 180,E1 14615.123,E2 14615.123} C_VEL
LIN {X 0,Y 315.04,Z 176.118,A -85,B 0,C 180,E1 14612.49,E2 14612.49} C_VEL
LIN {X 0,Y 308.18,Z 166.565,A -85,B 0,C 180,E1 14610.19,E2 14610.19} C_VEL
LIN {X 0,Y 303.939,Z 158.095,A -85,B 0,C 180,E1 14606.999,E2 14606.999} C_VEL
LIN {X 0,Y 301.355,Z 153.291,A -85,B 0,C 180,E1 14604.921,E2 14604.921} C_VEL
LIN {X 0,Y 299.005,Z 148.784,A -85,B 0,C 180,E1 14602.823,E2 14602.823} C_VEL
LIN {X 0,Y 296.758,Z 144.817,A -85,B 0,C 180,E1 14600.718,E2 14600.718} C_VEL
LIN {X 0,Y 295.968,Z 143.505,A -85,B 0,C 180,E1 14599.95,E2 14599.95} C_VEL
LIN {X 0,Y 293.856,Z 139.938,A -85,B 0,C 180,E1 14597.695,E2 14597.695} C_VEL
LIN {X 0,Y 293.223,Z 138.538,A -85,B 0,C 180,E1 14596.848,E2 14596.848} C_VEL
LIN {X 0,Y 290.742,Z 135.045,A -85,B 0,C 180,E1 14593.929,E2 14593.929} C_VEL
LIN {X 0,Y 290.316,Z 133.282,A -85,B 0,C 180,E1 14592.733,E2 14592.733} C_VEL
LIN {X 0,Y 290.321,Z 133.284,A -85,B 0,C 180,E1 14588.117,E2 14588.117} C_VEL
LIN {X 0,Y 290.302,Z 133.318,A -85,B 0,C 180,E1 14583.554,E2 14583.554} C_VEL
LIN {X 0,Y 290.304,Z 133.298,A -85,B 0,C 180,E1 14579.013,E2 14579.013} C_VEL
LIN {X 0,Y 290.324,Z 133.277,A -85,B 0,C 180,E1 14574.426,E2 14574.426} C_VEL
LIN {X 0,Y 290.301,Z 133.294,A -85,B 0,C 180,E1 14569.883,E2 14569.883} C_VEL
LIN {X 0,Y 290.302,Z 133.326,A -85,B 0,C 180,E1 14565.234,E2 14565.234} C_VEL
LIN {X 0,Y 290.345,Z 133.474,A -85,B 0,C 180,E1 14562.566,E2 14562.566} C_VEL
LIN {X 0,Y 291.993,Z 137.334,A -85,B 0,C 180,E1 14559.755,E2 14559.755} C_VEL
LIN {X 0,Y 293.493,Z 139.084,A -85,B 0,C 180,E1 14558.202,E2 14558.202} C_VEL
LIN {X 0,Y 295.385,Z 142.976,A -85,B 0,C 180,E1 14555.821,E2 14555.821} C_VEL
LIN {X 0,Y 296.274,Z 144.026,A -85,B 0,C 180,E1 14555.048,E2 14555.048} C_VEL
LIN {X 0,Y 298.055,Z 147.825,A -85,B 0,C 180,E1 14553.071,E2 14553.071} C_VEL
LIN {X 0,Y 298.941,Z 149.201,A -85,B 0,C 180,E1 14552.295,E2 14552.295} C_VEL
LIN {X 0,Y 301.635,Z 154.67,A -85,B 0,C 180,E1 14549.745,E2 14549.745} C_VEL
LIN {X 0,Y 303.978,Z 159.461,A -85,B 0,C 180,E1 14547.705,E2 14547.705} C_VEL
LIN {X 0,Y 307.537,Z 166.79,A -85,B 0,C 180,E1 14544.868,E2 14544.868} C_VEL
LIN {X 0,Y 309.745,Z 171.603,A -85,B 0,C 180,E1 14543.274,E2 14543.274} C_VEL
LIN {X 0,Y 318.513,Z 184.197,A -85,B 0,C 180,E1 14540.529,E2 14540.529} C_VEL
LIN {X 0,Y 327.652,Z 198.685,A -85,B 0,C 180,E1 14537.946,E2 14537.946} C_VEL
LIN {X 0,Y 336.166,Z 213.518,A -85,B 0,C 180,E1 14535.745,E2 14535.745} C_VEL
LIN {X 0,Y 341.806,Z 224.508,A -85,B 0,C 180,E1 14534.366,E2 14534.366} C_VEL
LIN {X 0,Y 341.948,Z 228.832,A -85,B 0,C 180,E1 14534.215,E2 14534.215} C_VEL
LIN {X 0,Y 334.33,Z 396.627,A -85,B 0,C 180,E1 14530.809,E2 14530.809} C_VEL
LIN {X 0,Y 332.486,Z 416.216,A -85,B 0,C 180,E1 14530.125,E2 14530.125} C_VEL
LIN {X 0,Y 329.936,Z 434.697,A -85,B 0,C 180,E1 14529.185,E2 14529.185} C_VEL
LIN {X 0,Y 326.699,Z 452.593,A -85,B 0,C 180,E1 14527.962,E2 14527.962} C_VEL
LIN {X 0,Y 322.721,Z 470.396,A -85,B 0,C 180,E1 14526.39,E2 14526.39} C_VEL
LIN {X 0,Y 318.362,Z 487.004,A -85,B 0,C 180,E1 14524.532,E2 14524.532} C_VEL
LIN {X 0,Y 313.742,Z 502.484,A -85,B 0,C 180,E1 14522.369,E2 14522.369} C_VEL
LIN {X 0,Y 308.977,Z 516.954,A -85,B 0,C 180,E1 14519.858,E2 14519.858} C_VEL
LIN {X 0,Y 304.536,Z 529.576,A -85,B 0,C 180,E1 14517.151,E2 14517.151} C_VEL
LIN {X 0,Y 300.405,Z 540.836,A -85,B 0,C 180,E1 14514.165,E2 14514.165} C_VEL
LIN {X 0,Y 296.574,Z 551.133,A -85,B 0,C 180,E1 14510.73,E2 14510.73} C_VEL
LIN {X 0,Y 293.609,Z 559.345,A -85,B 0,C 180,E1 14507.232,E2 14507.232} C_VEL
LIN {X 0,Y 291.341,Z 566.031,A -85,B 0,C 180,E1 14503.494,E2 14503.494} C_VEL
LIN {X 0,Y 289.882,Z 570.909,A -85,B 0,C 180,E1 14499.729,E2 14499.729} C_VEL
LIN {X 0,Y 289.036,Z 574.232,A -85,B 0,C 180,E1 14495.756,E2 14495.756} C_VEL
LIN {X 0,Y 288.709,Z 575.835,A -85,B 0,C 180,E1 14491.785,E2 14491.785} C_VEL
LIN {X 0,Y 288.715,Z 575.826,A -85,B 0,C 180,E1 14488.014,E2 14488.014} C_VEL
LIN {X 0,Y 289.054,Z 574.188,A -85,B 0,C 180,E1 14484.042,E2 14484.042} C_VEL
LIN {X 0,Y 289.92,Z 570.821,A -85,B 0,C 180,E1 14480.069,E2 14480.069} C_VEL
LIN {X 0,Y 291.51,Z 565.569,A -85,B 0,C 180,E1 14476.091,E2 14476.091} C_VEL
LIN {X 0,Y 293.911,Z 558.549,A -85,B 0,C 180,E1 14472.277,E2 14472.277} C_VEL
LIN {X 0,Y 296.886,Z 550.392,A -85,B 0,C 180,E1 14468.877,E2 14468.877} C_VEL
LIN {X 0,Y 300.554,Z 540.542,A -85,B 0,C 180,E1 14465.636,E2 14465.636} C_VEL
LIN {X 0,Y 304.716,Z 529.224,A -85,B 0,C 180,E1 14462.652,E2 14462.652} C_VEL
LIN {X 0,Y 309.231,Z 516.402,A -85,B 0,C 180,E1 14459.921,E2 14459.921} C_VEL
LIN {X 0,Y 313.973,Z 501.961,A -85,B 0,C 180,E1 14457.439,E2 14457.439} C_VEL
LIN {X 0,Y 318.595,Z 486.429,A -85,B 0,C 180,E1 14455.287,E2 14455.287} C_VEL
LIN {X 0,Y 322.993,Z 469.59,A -85,B 0,C 180,E1 14453.422,E2 14453.422} C_VEL
LIN {X 0,Y 326.773,Z 452.662,A -85,B 0,C 180,E1 14451.934,E2 14451.934} C_VEL
LIN {X 0,Y 330.124,Z 434.076,A -85,B 0,C 180,E1 14450.67,E2 14450.67} C_VEL
LIN {X 0,Y 331.515,Z 424.642,A -85,B 0,C 180,E1 14450.159,E2 14450.159} C_VEL
LIN {X 0,Y 331.73,Z 417.336,A -85,B 0,C 180,E1 14449.701,E2 14449.701} C_VEL
LIN {X 0,Y 329.259,Z 400.104,A -85,B 0,C 180,E1 14448.379,E2 14448.379} C_VEL
LIN {X 0,Y 328.908,Z 392.639,A -85,B 0,C 180,E1 14448.025,E2 14448.025} C_VEL
LIN {X 0,Y 328.948,Z 391.546,A -85,B 0,C 180,E1 14447.996,E2 14447.996} C_VEL
LIN {X 0,Y 336.568,Z 227.853,A -85,B 0,C 180,E1 14444.635,E2 14444.635} C_VEL
LIN {X 0,Y 327.851,Z 211.452,A -85,B 0,C 180,E1 14442.376,E2 14442.376} C_VEL
LIN {X 0,Y 324.592,Z 216.071,A -85,B 0,C 180,E1 14441.829,E2 14441.829} C_VEL
LIN {X 0,Y 323.596,Z 217.326,A -85,B 0,C 180,E1 14441.653,E2 14441.653} C_VEL
LIN {X 0,Y 317.896,Z 237.515,A -85,B 0,C 180,E1 14441.054,E2 14441.054} C_VEL
LIN {X 0,Y 314.754,Z 245.617,A -85,B 0,C 180,E1 14440.606,E2 14440.606} C_VEL
LIN {X 0,Y 313.08,Z 247.983,A -85,B 0,C 180,E1 14440.294,E2 14440.294} C_VEL
LIN {X 0,Y 312.14,Z 247.926,A -85,B 0,C 180,E1 14440.058,E2 14440.058} C_VEL
LIN {X 0,Y 301.839,Z 404.874,A -85,B 0,C 180,E1 14435.023,E2 14435.023} C_VEL
LIN {X 0,Y 300.244,Z 425.02,A -85,B 0,C 180,E1 14434.019,E2 14434.019} C_VEL
LIN {X 0,Y 298.205,Z 444.775,A -85,B 0,C 180,E1 14432.672,E2 14432.672} C_VEL
LIN {X 0,Y 295.892,Z 463.561,A -85,B 0,C 180,E1 14431.019,E2 14431.019} C_VEL
LIN {X 0,Y 293.403,Z 481.433,A -85,B 0,C 180,E1 14429.053,E2 14429.053} C_VEL
LIN {X 0,Y 290.836,Z 498.259,A -85,B 0,C 180,E1 14426.767,E2 14426.767} C_VEL
LIN {X 0,Y 288.386,Z 513.485,A -85,B 0,C 180,E1 14424.237,E2 14424.237} C_VEL
LIN {X 0,Y 286.206,Z 527.009,A -85,B 0,C 180,E1 14421.52,E2 14421.52} C_VEL
LIN {X 0,Y 284.258,Z 539.591,A -85,B 0,C 180,E1 14418.456,E2 14418.456} C_VEL
LIN {X 0,Y 282.794,Z 549.943,A -85,B 0,C 180,E1 14415.378,E2 14415.378} C_VEL
LIN {X 0,Y 281.713,Z 558.9,A -85,B 0,C 180,E1 14412.088,E2 14412.088} C_VEL
LIN {X 0,Y 281.027,Z 566.357,A -85,B 0,C 180,E1 14408.594,E2 14408.594} C_VEL
LIN {X 0,Y 280.711,Z 571.924,A -85,B 0,C 180,E1 14405.109,E2 14405.109} C_VEL
LIN {X 0,Y 280.671,Z 575.776,A -85,B 0,C 180,E1 14401.634,E2 14401.634} C_VEL
LIN {X 0,Y 280.862,Z 578.017,A -85,B 0,C 180,E1 14398.164,E2 14398.164} C_VEL
LIN {X 0,Y 281.373,Z 578.679,A -85,B 0,C 180,E1 14394.495,E2 14394.495} C_VEL
LIN {X 0,Y 282.352,Z 577.616,A -85,B 0,C 180,E1 14390.831,E2 14390.831} C_VEL
LIN {X 0,Y 283.943,Z 574.829,A -85,B 0,C 180,E1 14387.183,E2 14387.183} C_VEL
LIN {X 0,Y 286.291,Z 570.282,A -85,B 0,C 180,E1 14383.568,E2 14383.568} C_VEL
LIN {X 0,Y 289.669,Z 563.431,A -85,B 0,C 180,E1 14379.808,E2 14379.808} C_VEL
LIN {X 0,Y 293.802,Z 554.918,A -85,B 0,C 180,E1 14376.324,E2 14376.324} C_VEL
LIN {X 0,Y 298.559,Z 544.806,A -85,B 0,C 180,E1 14373.121,E2 14373.121} C_VEL
LIN {X 0,Y 304.163,Z 532.424,A -85,B 0,C 180,E1 14370.023,E2 14370.023} C_VEL
LIN {X 0,Y 310.27,Z 518.486,A -85,B 0,C 180,E1 14367.222,E2 14367.222} C_VEL
LIN {X 0,Y 316.747,Z 502.987,A -85,B 0,C 180,E1 14364.714,E2 14364.714} C_VEL
LIN {X 0,Y 323.788,Z 485.311,A -85,B 0,C 180,E1 14362.419,E2 14362.419} C_VEL
LIN {X 0,Y 330.5,Z 467.279,A -85,B 0,C 180,E1 14360.557,E2 14360.557} C_VEL
LIN {X 0,Y 336.953,Z 448.321,A -85,B 0,C 180,E1 14359.021,E2 14359.021} C_VEL
LIN {X 0,Y 342.611,Z 429.28,A -85,B 0,C 180,E1 14357.839,E2 14357.839} C_VEL
LIN {X 0,Y 343.613,Z 425.441,A -85,B 0,C 180,E1 14357.625,E2 14357.625} C_VEL
LIN {X 0,Y 334.604,Z 451.13,A -85,B 0,C 180,E1 14356.316,E2 14356.316} C_VEL
LIN {X 0,Y 327.857,Z 468.371,A -85,B 0,C 180,E1 14355.035,E2 14355.035} C_VEL
LIN {X 0,Y 320.2,Z 487.068,A -85,B 0,C 180,E1 14353.318,E2 14353.318} C_VEL
LIN {X 0,Y 310.368,Z 511.477,A -85,B 0,C 180,E1 14350.357,E2 14350.357} C_VEL
LIN {X 0,Y 303.002,Z 532.045,A -85,B 0,C 180,E1 14347.28,E2 14347.28} C_VEL
LIN {X 0,Y 298.142,Z 547.833,A -85,B 0,C 180,E1 14344.635,E2 14344.635} C_VEL
LIN {X 0,Y 293.766,Z 561.607,A -85,B 0,C 180,E1 14341.842,E2 14341.842} C_VEL
LIN {X 0,Y 289.491,Z 575.32,A -85,B 0,C 180,E1 14338.467,E2 14338.467} C_VEL
LIN {X 0,Y 285.923,Z 587.414,A -85,B 0,C 180,E1 14334.813,E2 14334.813} C_VEL
LIN {X 0,Y 283.2,Z 597.88,A -85,B 0,C 180,E1 14330.892,E2 14330.892} C_VEL
LIN {X 0,Y 281.455,Z 606.278,A -85,B 0,C 180,E1 14326.937,E2 14326.937} C_VEL
LIN {X 0,Y 280.536,Z 612.81,A -85,B 0,C 180,E1 14322.977,E2 14322.977} C_VEL
LIN {X 0,Y 280.269,Z 617.578,A -85,B 0,C 180,E1 14319.032,E2 14319.032} C_VEL
LIN {X 0,Y 280.348,Z 620.453,A -85,B 0,C 180,E1 14315.322,E2 14315.322} C_VEL
LIN {X 0,Y 280.48,Z 621.882,A -85,B 0,C 180,E1 14311.636,E2 14311.636} C_VEL
LIN {X 0,Y 280.481,Z 621.88,A -85,B 0,C 180,E1 14308.367,E2 14308.367} C_VEL
LIN {X 0,Y 280.35,Z 620.443,A -85,B 0,C 180,E1 14304.681,E2 14304.681} C_VEL
LIN {X 0,Y 280.27,Z 617.561,A -85,B 0,C 180,E1 14300.97,E2 14300.97} C_VEL
LIN {X 0,Y 280.537,Z 612.795,A -85,B 0,C 180,E1 14297.026,E2 14297.026} C_VEL
LIN {X 0,Y 281.452,Z 606.254,A -85,B 0,C 180,E1 14293.065,E2 14293.065} C_VEL
LIN {X 0,Y 283.196,Z 597.844,A -85,B 0,C 180,E1 14289.11,E2 14289.11} C_VEL
LIN {X 0,Y 285.748,Z 587.974,A -85,B 0,C 180,E1 14285.395,E2 14285.395} C_VEL
LIN {X 0,Y 289.109,Z 576.492,A -85,B 0,C 180,E1 14281.871,E2 14281.871} C_VEL
LIN {X 0,Y 292.941,Z 564.182,A -85,B 0,C 180,E1 14278.75,E2 14278.75} C_VEL
LIN {X 0,Y 297.656,Z 549.275,A -85,B 0,C 180,E1 14275.646,E2 14275.646} C_VEL
LIN {X 0,Y 302.425,Z 533.843,A -85,B 0,C 180,E1 14273.009,E2 14273.009} C_VEL
LIN {X 0,Y 307.425,Z 516.844,A -85,B 0,C 180,E1 14270.64,E2 14270.64} C_VEL
LIN {X 0,Y 312.277,Z 498.859,A -85,B 0,C 180,E1 14268.612,E2 14268.612} C_VEL
LIN {X 0,Y 316.753,Z 480.208,A -85,B 0,C 180,E1 14266.929,E2 14266.929} C_VEL
